gfCNCPoint4[10892] = {X 149.4831, Y 49.3200, Z -5.5000, A 0.000, B 0.000, C 0.000 }
gfCNCPoint4[10893] = {X 143.0396, Y 49.3200, Z -5.5000, A 0.000, B 0.000, C 0.000 }
gfCNCPoint4[10894] = {X 142.0831, Y 49.2128, Z -5.5000, A 0.000, B 0.000, C 0.000 }
gfCNCPoint4[10895] = {X 141.1741, Y 48.8964, Z -5.5000, A 0.000, B 0.000, C 0.000 }
gfCNCPoint4[10896] = {X 140.3576, Y 48.3866, Z -5.5000, A 0.000, B 0.000, C 0.000 }
gfCNCPoint4[10897] = {X 139.6743, Y 47.7087, Z -5.5000, A 0.000, B 0.000, C 0.000 }
gfCNCPoint4[10898] = {X 139.1581, Y 46.8964, Z -5.5000, A 0.000, B 0.000, C 0.000 }
gfCNCPoint4[10899] = {X 138.8346, Y 45.9899, Z -5.5000, A 0.000, B 0.000, C 0.000 }
gfCNCPoint4[10900] = {X 138.7198, Y 45.0342, Z -5.5000, A 0.000, B 0.000, C 0.000 }
gfCNCPoint4[10901] = {X 138.7200, Y 44.1494, Z -5.5000, A 0.000, B 0.000, C 0.000 }
gfCNCPoint4[10902] = {X 138.8305, Y 43.2364, Z -5.5000, A 0.000, B 0.000, C 0.000 }
gfCNCPoint4[10903] = {X 139.1317, Y 42.3675, Z -5.5000, A 0.000, B 0.000, C 0.000 }
gfCNCPoint4[10904] = {X 139.6099, Y 41.5821, Z -5.5000, A 0.000, B 0.000, C 0.000 }
gfCNCPoint4[10905] = {X 140.2436, Y 40.9157, Z -5.5000, A 0.000, B 0.000, C 0.000 }
gfCNCPoint4[10906] = {X 140.2436, Y 30.3967, Z -5.5000, A 0.000, B 0.000, C 0.000 }
gfCNCPoint4[10907] = {X 136.2436, Y 30.3967, Z -5.5000, A 0.000, B 0.000, C 0.000 }
gfCNCPoint4[10908] = {X 140.3236, Y 30.3967, Z -5.5000, A 0.000, B 0.000, C 0.000 }
gfCNCPoint4[10909] = {X 140.3236, Y 19.7977, Z -5.5000, A 0.000, B 0.000, C 0.000 }
gfCNCPoint4[10910] = {X 137.3795, Y 19.7972, Z -5.5000, A 0.000, B 0.000, C 0.000 }
gfCNCPoint4[10911] = {X 137.3567, Y 19.8337, Z -5.5000, A 0.000, B 0.000, C 0.000 }
gfCNCPoint4[10912] = {X 136.8341, Y 20.4660, Z -5.5000, A 0.000, B 0.000, C 0.000 }
gfCNCPoint4[10913] = {X 136.1996, Y 20.9859, Z -5.5000, A 0.000, B 0.000, C 0.000 }
gfCNCPoint4[10914] = {X 135.4768, Y 21.3738, Z -5.5000, A 0.000, B 0.000, C 0.000 }
gfCNCPoint4[10915] = {X 134.6929, Y 21.6153, Z -5.5000, A 0.000, B 0.000, C 0.000 }
gfCNCPoint4[10916] = {X 133.8772, Y 21.7014, Z -5.5000, A 0.000, B 0.000, C 0.000 }
gfCNCPoint4[10917] = {X 133.2006, Y 21.7015, Z -5.5000, A 0.000, B 0.000, C 0.000 }
gfCNCPoint4[10918] = {X 132.2572, Y 21.5952, Z -5.5000, A 0.000, B 0.000, C 0.000 }
gfCNCPoint4[10919] = {X 131.3610, Y 21.2816, Z -5.5000, A 0.000, B 0.000, C 0.000 }
gfCNCPoint4[10920] = {X 130.5570, Y 20.7765, Z -5.5000, A 0.000, B 0.000, C 0.000 }
gfCNCPoint4[10921] = {X 129.8857, Y 20.1051, Z -5.5000, A 0.000, B 0.000, C 0.000 }
gfCNCPoint4[10922] = {X 129.3805, Y 19.3012, Z -5.5000, A 0.000, B 0.000, C 0.000 }
gfCNCPoint4[10923] = {X 129.0669, Y 18.4050, Z -5.5000, A 0.000, B 0.000, C 0.000 }
gfCNCPoint4[10924] = {X 128.9606, Y 17.4615, Z -5.5000, A 0.000, B 0.000, C 0.000 }
gfCNCPoint4[10925] = {X 128.9606, Y 10.4835, Z -5.5000, A 0.000, B 0.000, C 0.000 }
gfCNCPoint4[10926] = {X 129.0655, Y 9.5466, Z -5.5000, A 0.000, B 0.000, C 0.000 }
gfCNCPoint4[10927] = {X 129.3747, Y 8.6559, Z -5.5000, A 0.000, B 0.000, C 0.000 }
gfCNCPoint4[10928] = {X 129.8732, Y 7.8557, Z -5.5000, A 0.000, B 0.000, C 0.000 }
gfCNCPoint4[10929] = {X 130.5362, Y 7.1853, Z -5.5000, A 0.000, B 0.000, C 0.000 }
gfCNCPoint4[10930] = {X 131.3309, Y 6.6781, Z -5.5000, A 0.000, B 0.000, C 0.000 }
gfCNCPoint4[10931] = {X 132.2180, Y 6.3589, Z -5.5000, A 0.000, B 0.000, C 0.000 }
gfCNCPoint4[10932] = {X 133.1538, Y 6.2438, Z -5.5000, A 0.000, B 0.000, C 0.000 }
gfCNCPoint4[10933] = {X 133.8858, Y 6.2437, Z -5.5000, A 0.000, B 0.000, C 0.000 }
gfCNCPoint4[10934] = {X 134.7031, Y 6.3318, Z -5.5000, A 0.000, B 0.000, C 0.000 }
gfCNCPoint4[10935] = {X 135.4881, Y 6.5760, Z -5.5000, A 0.000, B 0.000, C 0.000 }
gfCNCPoint4[10936] = {X 136.2112, Y 6.9670, Z -5.5000, A 0.000, B 0.000, C 0.000 }
gfCNCPoint4[10937] = {X 136.8453, Y 7.4903, Z -5.5000, A 0.000, B 0.000, C 0.000 }
gfCNCPoint4[10938] = {X 137.3665, Y 8.1260, Z -5.5000, A 0.000, B 0.000, C 0.000 }
gfCNCPoint4[10939] = {X 155.1554, Y 8.1273, Z -5.5000, A 0.000, B 0.000, C 0.000 }
gfCNCPoint4[10940] = {X 155.6773, Y 7.4904, Z -5.5000, A 0.000, B 0.000, C 0.000 }
gfCNCPoint4[10941] = {X 156.3124, Y 6.9664, Z -5.5000, A 0.000, B 0.000, C 0.000 }
gfCNCPoint4[10942] = {X 157.0368, Y 6.5750, Z -5.5000, A 0.000, B 0.000, C 0.000 }
gfCNCPoint4[10943] = {X 157.8232, Y 6.3311, Z -5.5000, A 0.000, B 0.000, C 0.000 }
gfCNCPoint4[10944] = {X 158.6420, Y 6.2437, Z -5.5000, A 0.000, B 0.000, C 0.000 }
gfCNCPoint4[10945] = {X 159.3770, Y 6.2439, Z -5.5000, A 0.000, B 0.000, C 0.000 }
gfCNCPoint4[10946] = {X 160.3114, Y 6.3606, Z -5.5000, A 0.000, B 0.000, C 0.000 }
gfCNCPoint4[10947] = {X 161.1970, Y 6.6806, Z -5.5000, A 0.000, B 0.000, C 0.000 }
gfCNCPoint4[10948] = {X 161.9902, Y 7.1882, Z -5.5000, A 0.000, B 0.000, C 0.000 }
gfCNCPoint4[10949] = {X 162.6517, Y 7.8584, Z -5.5000, A 0.000, B 0.000, C 0.000 }
gfCNCPoint4[10950] = {X 163.1490, Y 8.6580, Z -5.5000, A 0.000, B 0.000, C 0.000 }
gfCNCPoint4[10951] = {X 163.4575, Y 9.5477, Z -5.5000, A 0.000, B 0.000, C 0.000 }
gfCNCPoint4[10952] = {X 163.5621, Y 10.4835, Z -5.5000, A 0.000, B 0.000, C 0.000 }
gfCNCPoint4[10953] = {X 163.5621, Y 17.4615, Z -5.5000, A 0.000, B 0.000, C 0.000 }
gfCNCPoint4[10954] = {X 163.4575, Y 18.3975, Z -5.5000, A 0.000, B 0.000, C 0.000 }
gfCNCPoint4[10955] = {X 163.1489, Y 19.2873, Z -5.5000, A 0.000, B 0.000, C 0.000 }
gfCNCPoint4[10956] = {X 162.6514, Y 20.0870, Z -5.5000, A 0.000, B 0.000, C 0.000 }
gfCNCPoint4[10957] = {X 161.9897, Y 20.7572, Z -5.5000, A 0.000, B 0.000, C 0.000 }
gfCNCPoint4[10958] = {X 161.1964, Y 21.2648, Z -5.5000, A 0.000, B 0.000, C 0.000 }
gfCNCPoint4[10959] = {X 160.3106, Y 21.5847, Z -5.5000, A 0.000, B 0.000, C 0.000 }
gfCNCPoint4[10960] = {X 159.3760, Y 21.7012, Z -5.5000, A 0.000, B 0.000, C 0.000 }
gfCNCPoint4[10961] = {X 158.6796, Y 21.7015, Z -5.5000, A 0.000, B 0.000, C 0.000 }
gfCNCPoint4[10962] = {X 157.8483, Y 21.6166, Z -5.5000, A 0.000, B 0.000, C 0.000 }
gfCNCPoint4[10963] = {X 157.0495, Y 21.3715, Z -5.5000, A 0.000, B 0.000, C 0.000 }
gfCNCPoint4[10964] = {X 156.3137, Y 20.9756, Z -5.5000, A 0.000, B 0.000, C 0.000 }
gfCNCPoint4[10965] = {X 155.6689, Y 20.4441, Z -5.5000, A 0.000, B 0.000, C 0.000 }
gfCNCPoint4[10966] = {X 155.1400, Y 19.7973, Z -5.5000, A 0.000, B 0.000, C 0.000 }
gfCNCPoint4[10967] = {X 152.1967, Y 19.7984, Z -5.5000, A 0.000, B 0.000, C 0.000 }
gfCNCPoint4[10968] = {X 152.1954, Y 40.9056, Z -5.5000, A 0.000, B 0.000, C 0.000 }
gfCNCPoint4[10969] = {X 152.6809, Y 41.4282, Z -5.5000, A 0.000, B 0.000, C 0.000 }
gfCNCPoint4[10970] = {X 152.7744, Y 41.5396, Z -5.5000, A 0.000, B 0.000, C 0.000 }
gfCNCPoint4[10971] = {X 153.2900, Y 42.3496, Z -5.5000, A 0.000, B 0.000, C 0.000 }
gfCNCPoint4[10972] = {X 153.6117, Y 43.2543, Z -5.5000, A 0.000, B 0.000, C 0.000 }
gfCNCPoint4[10973] = {X 153.7231, Y 44.2080, Z -5.5000, A 0.000, B 0.000, C 0.000 }
gfCNCPoint4[10974] = {X 153.7229, Y 45.0408, Z -5.5000, A 0.000, B 0.000, C 0.000 }
gfCNCPoint4[10975] = {X 153.6089, Y 45.9775, Z -5.5000, A 0.000, B 0.000, C 0.000 }
gfCNCPoint4[10976] = {X 153.2905, Y 46.8659, Z -5.5000, A 0.000, B 0.000, C 0.000 }
gfCNCPoint4[10977] = {X 152.7835, Y 47.6618, Z -5.5000, A 0.000, B 0.000, C 0.000 }
gfCNCPoint4[10978] = {X 152.1130, Y 48.3258, Z -5.5000, A 0.000, B 0.000, C 0.000 }
gfCNCPoint4[10979] = {X 151.3123, Y 48.8251, Z -5.5000, A 0.000, B 0.000, C 0.000 }
gfCNCPoint4[10980] = {X 150.4209, Y 49.1350, Z -5.5000, A 0.000, B 0.000, C 0.000 }
gfCNCPoint4[10981] = {X 149.4831, Y 49.2400, Z -5.5000, A 0.000, B 0.000, C 0.000 }
gfCNCPoint4[10982] = {X 143.0396, Y 49.2400, Z -5.5000, A 0.000, B 0.000, C 0.000 }
gfCNCPoint4[10983] = {X 142.1008, Y 49.1348, Z -5.5000, A 0.000, B 0.000, C 0.000 }
gfCNCPoint4[10984] = {X 141.2086, Y 48.8243, Z -5.5000, A 0.000, B 0.000, C 0.000 }
gfCNCPoint4[10985] = {X 140.4073, Y 48.3239, Z -5.5000, A 0.000, B 0.000, C 0.000 }
gfCNCPoint4[10986] = {X 139.7367, Y 47.6586, Z -5.5000, A 0.000, B 0.000, C 0.000 }
gfCNCPoint4[10987] = {X 139.2300, Y 46.8612, Z -5.5000, A 0.000, B 0.000, C 0.000 }
gfCNCPoint4[10988] = {X 138.9124, Y 45.9715, Z -5.5000, A 0.000, B 0.000, C 0.000 }
gfCNCPoint4[10989] = {X 138.7998, Y 45.0336, Z -5.5000, A 0.000, B 0.000, C 0.000 }
gfCNCPoint4[10990] = {X 138.8000, Y 44.1505, Z -5.5000, A 0.000, B 0.000, C 0.000 }
gfCNCPoint4[10991] = {X 138.9105, Y 43.2454, Z -5.5000, A 0.000, B 0.000, C 0.000 }
gfCNCPoint4[10992] = {X 139.2119, Y 42.3850, Z -5.5000, A 0.000, B 0.000, C 0.000 }
gfCNCPoint4[10993] = {X 139.6903, Y 41.6088, Z -5.5000, A 0.000, B 0.000, C 0.000 }
gfCNCPoint4[10994] = {X 140.3236, Y 40.9529, Z -5.5000, A 0.000, B 0.000, C 0.000 }
gfCNCPoint4[10995] = {X 140.3236, Y 30.3967, Z -5.5000, A 0.000, B 0.000, C 0.000 }
gfCNCPoint4[10996] = {X 136.3236, Y 30.3967, Z -5.5000, A 0.000, B 0.000, C 0.000 }
gfCNCPoint4[10997] = {X 140.4036, Y 30.3967, Z -5.5000, A 0.000, B 0.000, C 0.000 }
gfCNCPoint4[10998] = {X 140.4036, Y 19.7178, Z -5.5000, A 0.000, B 0.000, C 0.000 }
gfCNCPoint4[10999] = {X 137.3353, Y 19.7172, Z -5.5000, A 0.000, B 0.000, C 0.000 }
gfCNCPoint4[11000] = {X 137.2896, Y 19.7900, Z -5.5000, A 0.000, B 0.000, C 0.000 }
gfCNCPoint4[11001] = {X 136.7769, Y 20.4101, Z -5.5000, A 0.000, B 0.000, C 0.000 }
gfCNCPoint4[11002] = {X 136.1544, Y 20.9198, Z -5.5000, A 0.000, B 0.000, C 0.000 }
gfCNCPoint4[11003] = {X 135.4455, Y 21.3002, Z -5.5000, A 0.000, B 0.000, C 0.000 }
gfCNCPoint4[11004] = {X 134.6766, Y 21.5370, Z -5.5000, A 0.000, B 0.000, C 0.000 }
gfCNCPoint4[11005] = {X 133.8765, Y 21.6214, Z -5.5000, A 0.000, B 0.000, C 0.000 }
gfCNCPoint4[11006] = {X 133.2006, Y 21.6215, Z -5.5000, A 0.000, B 0.000, C 0.000 }
gfCNCPoint4[11007] = {X 132.2750, Y 21.5172, Z -5.5000, A 0.000, B 0.000, C 0.000 }
gfCNCPoint4[11008] = {X 131.3957, Y 21.2096, Z -5.5000, A 0.000, B 0.000, C 0.000 }
gfCNCPoint4[11009] = {X 130.6069, Y 20.7140, Z -5.5000, A 0.000, B 0.000, C 0.000 }
gfCNCPoint4[11010] = {X 129.9482, Y 20.0553, Z -5.5000, A 0.000, B 0.000, C 0.000 }
gfCNCPoint4[11011] = {X 129.4526, Y 19.2665, Z -5.5000, A 0.000, B 0.000, C 0.000 }
gfCNCPoint4[11012] = {X 129.1449, Y 18.3872, Z -5.5000, A 0.000, B 0.000, C 0.000 }
gfCNCPoint4[11013] = {X 129.0406, Y 17.4615, Z -5.5000, A 0.000, B 0.000, C 0.000 }
gfCNCPoint4[11014] = {X 129.0406, Y 10.4835, Z -5.5000, A 0.000, B 0.000, C 0.000 }
gfCNCPoint4[11015] = {X 129.1435, Y 9.5642, Z -5.5000, A 0.000, B 0.000, C 0.000 }
gfCNCPoint4[11016] = {X 129.4469, Y 8.6904, Z -5.5000, A 0.000, B 0.000, C 0.000 }
gfCNCPoint4[11017] = {X 129.9360, Y 7.9052, Z -5.5000, A 0.000, B 0.000, C 0.000 }
gfCNCPoint4[11018] = {X 130.5864, Y 7.2475, Z -5.5000, A 0.000, B 0.000, C 0.000 }
gfCNCPoint4[11019] = {X 131.3661, Y 6.7499, Z -5.5000, A 0.000, B 0.000, C 0.000 }
gfCNCPoint4[11020] = {X 132.2366, Y 6.4368, Z -5.5000, A 0.000, B 0.000, C 0.000 }
gfCNCPoint4[11021] = {X 133.1547, Y 6.3238, Z -5.5000, A 0.000, B 0.000, C 0.000 }
gfCNCPoint4[11022] = {X 133.8850, Y 6.3237, Z -5.5000, A 0.000, B 0.000, C 0.000 }
gfCNCPoint4[11023] = {X 134.6952, Y 6.4119, Z -5.5000, A 0.000, B 0.000, C 0.000 }
gfCNCPoint4[11024] = {X 135.4728, Y 6.6563, Z -5.5000, A 0.000, B 0.000, C 0.000 }
gfCNCPoint4[11025] = {X 136.1877, Y 7.0477, Z -5.5000, A 0.000, B 0.000, C 0.000 }
gfCNCPoint4[11026] = {X 136.8126, Y 7.5710, Z -5.5000, A 0.000, B 0.000, C 0.000 }
gfCNCPoint4[11027] = {X 137.3235, Y 8.2060, Z -5.5000, A 0.000, B 0.000, C 0.000 }
gfCNCPoint4[11028] = {X 155.1984, Y 8.2073, Z -5.5000, A 0.000, B 0.000, C 0.000 }
gfCNCPoint4[11029] = {X 155.7100, Y 7.5711, Z -5.5000, A 0.000, B 0.000, C 0.000 }
gfCNCPoint4[11030] = {X 156.3359, Y 7.0471, Z -5.5000, A 0.000, B 0.000, C 0.000 }
gfCNCPoint4[11031] = {X 157.0521, Y 6.6554, Z -5.5000, A 0.000, B 0.000, C 0.000 }
gfCNCPoint4[11032] = {X 157.8310, Y 6.4111, Z -5.5000, A 0.000, B 0.000, C 0.000 }
gfCNCPoint4[11033] = {X 158.6427, Y 6.3237, Z -5.5000, A 0.000, B 0.000, C 0.000 }
gfCNCPoint4[11034] = {X 159.3760, Y 6.3239, Z -5.5000, A 0.000, B 0.000, C 0.000 }
gfCNCPoint4[11035] = {X 160.2928, Y 6.4383, Z -5.5000, A 0.000, B 0.000, C 0.000 }
gfCNCPoint4[11036] = {X 161.1617, Y 6.7524, Z -5.5000, A 0.000, B 0.000, C 0.000 }
gfCNCPoint4[11037] = {X 161.9398, Y 7.2504, Z -5.5000, A 0.000, B 0.000, C 0.000 }
gfCNCPoint4[11038] = {X 162.5889, Y 7.9079, Z -5.5000, A 0.000, B 0.000, C 0.000 }
gfCNCPoint4[11039] = {X 163.0768, Y 8.6925, Z -5.5000, A 0.000, B 0.000, C 0.000 }
gfCNCPoint4[11040] = {X 163.3795, Y 9.5653, Z -5.5000, A 0.000, B 0.000, C 0.000 }
gfCNCPoint4[11041] = {X 163.4821, Y 10.4835, Z -5.5000, A 0.000, B 0.000, C 0.000 }
gfCNCPoint4[11042] = {X 163.4821, Y 17.4615, Z -5.5000, A 0.000, B 0.000, C 0.000 }
gfCNCPoint4[11043] = {X 163.3795, Y 18.3798, Z -5.5000, A 0.000, B 0.000, C 0.000 }
gfCNCPoint4[11044] = {X 163.0767, Y 19.2527, Z -5.5000, A 0.000, B 0.000, C 0.000 }
gfCNCPoint4[11045] = {X 162.5887, Y 20.0373, Z -5.5000, A 0.000, B 0.000, C 0.000 }
gfCNCPoint4[11046] = {X 161.9396, Y 20.6948, Z -5.5000, A 0.000, B 0.000, C 0.000 }
gfCNCPoint4[11047] = {X 161.1613, Y 21.1929, Z -5.5000, A 0.000, B 0.000, C 0.000 }
gfCNCPoint4[11048] = {X 160.2923, Y 21.5068, Z -5.5000, A 0.000, B 0.000, C 0.000 }
gfCNCPoint4[11049] = {X 159.3755, Y 21.6212, Z -5.5000, A 0.000, B 0.000, C 0.000 }
gfCNCPoint4[11050] = {X 158.6799, Y 21.6215, Z -5.5000, A 0.000, B 0.000, C 0.000 }
gfCNCPoint4[11051] = {X 157.8558, Y 21.5365, Z -5.5000, A 0.000, B 0.000, C 0.000 }
gfCNCPoint4[11052] = {X 157.0646, Y 21.2910, Z -5.5000, A 0.000, B 0.000, C 0.000 }
gfCNCPoint4[11053] = {X 156.3370, Y 20.8948, Z -5.5000, A 0.000, B 0.000, C 0.000 }
gfCNCPoint4[11054] = {X 155.7016, Y 20.3633, Z -5.5000, A 0.000, B 0.000, C 0.000 }
gfCNCPoint4[11055] = {X 155.1830, Y 19.7172, Z -5.5000, A 0.000, B 0.000, C 0.000 }
gfCNCPoint4[11056] = {X 152.1167, Y 19.7184, Z -5.5000, A 0.000, B 0.000, C 0.000 }
gfCNCPoint4[11057] = {X 152.1154, Y 40.9370, Z -5.5000, A 0.000, B 0.000, C 0.000 }
gfCNCPoint4[11058] = {X 152.6209, Y 41.4812, Z -5.5000, A 0.000, B 0.000, C 0.000 }
gfCNCPoint4[11059] = {X 152.7126, Y 41.5905, Z -5.5000, A 0.000, B 0.000, C 0.000 }
gfCNCPoint4[11060] = {X 153.2184, Y 42.3852, Z -5.5000, A 0.000, B 0.000, C 0.000 }
gfCNCPoint4[11061] = {X 153.5338, Y 43.2727, Z -5.5000, A 0.000, B 0.000, C 0.000 }
gfCNCPoint4[11062] = {X 153.6431, Y 44.2083, Z -5.5000, A 0.000, B 0.000, C 0.000 }
gfCNCPoint4[11063] = {X 153.6429, Y 45.0400, Z -5.5000, A 0.000, B 0.000, C 0.000 }
gfCNCPoint4[11064] = {X 153.5310, Y 45.9591, Z -5.5000, A 0.000, B 0.000, C 0.000 }
gfCNCPoint4[11065] = {X 153.2186, Y 46.8306, Z -5.5000, A 0.000, B 0.000, C 0.000 }
gfCNCPoint4[11066] = {X 152.7212, Y 47.6115, Z -5.5000, A 0.000, B 0.000, C 0.000 }
gfCNCPoint4[11067] = {X 152.0634, Y 48.2631, Z -5.5000, A 0.000, B 0.000, C 0.000 }
gfCNCPoint4[11068] = {X 151.2778, Y 48.7530, Z -5.5000, A 0.000, B 0.000, C 0.000 }
gfCNCPoint4[11069] = {X 150.4032, Y 49.0570, Z -5.5000, A 0.000, B 0.000, C 0.000 }
gfCNCPoint4[11070] = {X 149.4831, Y 49.1600, Z -5.5000, A 0.000, B 0.000, C 0.000 }
gfCNCPoint4[11071] = {X 143.0396, Y 49.1600, Z -5.5000, A 0.000, B 0.000, C 0.000 }
gfCNCPoint4[11072] = {X 142.1185, Y 49.0567, Z -5.5000, A 0.000, B 0.000, C 0.000 }
gfCNCPoint4[11073] = {X 141.2432, Y 48.7521, Z -5.5000, A 0.000, B 0.000, C 0.000 }
gfCNCPoint4[11074] = {X 140.4570, Y 48.2612, Z -5.5000, A 0.000, B 0.000, C 0.000 }
gfCNCPoint4[11075] = {X 139.7990, Y 47.6084, Z -5.5000, A 0.000, B 0.000, C 0.000 }
gfCNCPoint4[11076] = {X 139.3019, Y 46.8261, Z -5.5000, A 0.000, B 0.000, C 0.000 }
gfCNCPoint4[11077] = {X 138.9903, Y 45.9532, Z -5.5000, A 0.000, B 0.000, C 0.000 }
gfCNCPoint4[11078] = {X 138.8798, Y 45.0329, Z -5.5000, A 0.000, B 0.000, C 0.000 }
gfCNCPoint4[11079] = {X 138.8800, Y 44.1516, Z -5.5000, A 0.000, B 0.000, C 0.000 }
gfCNCPoint4[11080] = {X 138.9906, Y 43.2545, Z -5.5000, A 0.000, B 0.000, C 0.000 }
gfCNCPoint4[11081] = {X 139.2922, Y 42.4026, Z -5.5000, A 0.000, B 0.000, C 0.000 }
gfCNCPoint4[11082] = {X 139.7708, Y 41.6358, Z -5.5000, A 0.000, B 0.000, C 0.000 }
gfCNCPoint4[11083] = {X 140.4036, Y 40.9906, Z -5.5000, A 0.000, B 0.000, C 0.000 }
gfCNCPoint4[11084] = {X 140.4036, Y 30.3967, Z -5.5000, A 0.000, B 0.000, C 0.000 }
gfCNCPoint4[11085] = {X 136.4036, Y 30.3967, Z -5.5000, A 0.000, B 0.000, C 0.000 }
gfCNCPoint4[11086] = {X 140.4836, Y 30.3967, Z -5.5000, A 0.000, B 0.000, C 0.000 }
gfCNCPoint4[11087] = {X 140.4836, Y 19.6378, Z -5.5000, A 0.000, B 0.000, C 0.000 }
gfCNCPoint4[11088] = {X 137.2910, Y 19.6372, Z -5.5000, A 0.000, B 0.000, C 0.000 }
gfCNCPoint4[11089] = {X 137.2218, Y 19.7475, Z -5.5000, A 0.000, B 0.000, C 0.000 }
gfCNCPoint4[11090] = {X 136.5756, Y 20.4907, Z -5.5000, A 0.000, B 0.000, C 0.000 }
gfCNCPoint4[11091] = {X 135.7702, Y 21.0573, Z -5.5000, A 0.000, B 0.000, C 0.000 }
gfCNCPoint4[11092] = {X 134.8524, Y 21.4145, Z -5.5000, A 0.000, B 0.000, C 0.000 }
gfCNCPoint4[11093] = {X 133.8758, Y 21.5414, Z -5.5000, A 0.000, B 0.000, C 0.000 }
gfCNCPoint4[11094] = {X 133.2006, Y 21.5415, Z -5.5000, A 0.000, B 0.000, C 0.000 }
gfCNCPoint4[11095] = {X 132.2928, Y 21.4392, Z -5.5000, A 0.000, B 0.000, C 0.000 }
gfCNCPoint4[11096] = {X 131.4304, Y 21.1375, Z -5.5000, A 0.000, B 0.000, C 0.000 }
gfCNCPoint4[11097] = {X 130.6568, Y 20.6514, Z -5.5000, A 0.000, B 0.000, C 0.000 }
gfCNCPoint4[11098] = {X 130.0108, Y 20.0054, Z -5.5000, A 0.000, B 0.000, C 0.000 }
gfCNCPoint4[11099] = {X 129.5247, Y 19.2318, Z -5.5000, A 0.000, B 0.000, C 0.000 }
gfCNCPoint4[11100] = {X 129.2229, Y 18.3694, Z -5.5000, A 0.000, B 0.000, C 0.000 }
gfCNCPoint4[11101] = {X 129.1206, Y 17.4615, Z -5.5000, A 0.000, B 0.000, C 0.000 }
gfCNCPoint4[11102] = {X 129.1206, Y 10.4835, Z -5.5000, A 0.000, B 0.000, C 0.000 }
gfCNCPoint4[11103] = {X 129.2215, Y 9.5820, Z -5.5000, A 0.000, B 0.000, C 0.000 }
gfCNCPoint4[11104] = {X 129.5191, Y 8.7250, Z -5.5000, A 0.000, B 0.000, C 0.000 }
gfCNCPoint4[11105] = {X 129.9986, Y 7.9550, Z -5.5000, A 0.000, B 0.000, C 0.000 }
gfCNCPoint4[11106] = {X 130.6365, Y 7.3099, Z -5.5000, A 0.000, B 0.000, C 0.000 }
gfCNCPoint4[11107] = {X 131.4011, Y 6.8218, Z -5.5000, A 0.000, B 0.000, C 0.000 }
gfCNCPoint4[11108] = {X 132.2547, Y 6.5147, Z -5.5000, A 0.000, B 0.000, C 0.000 }
gfCNCPoint4[11109] = {X 133.1551, Y 6.4038, Z -5.5000, A 0.000, B 0.000, C 0.000 }
gfCNCPoint4[11110] = {X 133.8841, Y 6.4037, Z -5.5000, A 0.000, B 0.000, C 0.000 }
gfCNCPoint4[11111] = {X 134.6873, Y 6.4920, Z -5.5000, A 0.000, B 0.000, C 0.000 }
gfCNCPoint4[11112] = {X 135.4573, Y 6.7367, Z -5.5000, A 0.000, B 0.000, C 0.000 }
gfCNCPoint4[11113] = {X 136.1639, Y 7.1284, Z -5.5000, A 0.000, B 0.000, C 0.000 }
gfCNCPoint4[11114] = {X 136.7795, Y 7.6517, Z -5.5000, A 0.000, B 0.000, C 0.000 }
gfCNCPoint4[11115] = {X 137.2800, Y 8.2860, Z -5.5000, A 0.000, B 0.000, C 0.000 }
gfCNCPoint4[11116] = {X 155.2419, Y 8.2873, Z -5.5000, A 0.000, B 0.000, C 0.000 }
gfCNCPoint4[11117] = {X 155.2874, Y 8.2177, Z -5.5000, A 0.000, B 0.000, C 0.000 }
gfCNCPoint4[11118] = {X 155.3342, Y 8.1491, Z -5.5000, A 0.000, B 0.000, C 0.000 }
gfCNCPoint4[11119] = {X 155.9794, Y 7.4256, Z -5.5000, A 0.000, B 0.000, C 0.000 }
gfCNCPoint4[11120] = {X 156.7770, Y 6.8747, Z -5.5000, A 0.000, B 0.000, C 0.000 }
gfCNCPoint4[11121] = {X 157.6820, Y 6.5276, Z -5.5000, A 0.000, B 0.000, C 0.000 }
gfCNCPoint4[11122] = {X 158.6434, Y 6.4037, Z -5.5000, A 0.000, B 0.000, C 0.000 }
gfCNCPoint4[11123] = {X 159.3750, Y 6.4039, Z -5.5000, A 0.000, B 0.000, C 0.000 }
gfCNCPoint4[11124] = {X 160.2741, Y 6.5161, Z -5.5000, A 0.000, B 0.000, C 0.000 }
gfCNCPoint4[11125] = {X 161.1263, Y 6.8241, Z -5.5000, A 0.000, B 0.000, C 0.000 }
gfCNCPoint4[11126] = {X 161.8895, Y 7.3126, Z -5.5000, A 0.000, B 0.000, C 0.000 }
gfCNCPoint4[11127] = {X 162.5260, Y 7.9574, Z -5.5000, A 0.000, B 0.000, C 0.000 }
gfCNCPoint4[11128] = {X 163.0046, Y 8.7269, Z -5.5000, A 0.000, B 0.000, C 0.000 }
gfCNCPoint4[11129] = {X 163.3015, Y 9.5830, Z -5.5000, A 0.000, B 0.000, C 0.000 }
gfCNCPoint4[11130] = {X 163.4021, Y 10.4835, Z -5.5000, A 0.000, B 0.000, C 0.000 }
gfCNCPoint4[11131] = {X 163.4021, Y 17.4615, Z -5.5000, A 0.000, B 0.000, C 0.000 }
gfCNCPoint4[11132] = {X 163.3015, Y 18.3621, Z -5.5000, A 0.000, B 0.000, C 0.000 }
gfCNCPoint4[11133] = {X 163.0046, Y 19.2182, Z -5.5000, A 0.000, B 0.000, C 0.000 }
gfCNCPoint4[11134] = {X 162.5260, Y 19.9876, Z -5.5000, A 0.000, B 0.000, C 0.000 }
gfCNCPoint4[11135] = {X 161.8895, Y 20.6325, Z -5.5000, A 0.000, B 0.000, C 0.000 }
gfCNCPoint4[11136] = {X 161.1263, Y 21.1209, Z -5.5000, A 0.000, B 0.000, C 0.000 }
gfCNCPoint4[11137] = {X 160.2741, Y 21.4289, Z -5.5000, A 0.000, B 0.000, C 0.000 }
gfCNCPoint4[11138] = {X 159.3750, Y 21.5412, Z -5.5000, A 0.000, B 0.000, C 0.000 }
gfCNCPoint4[11139] = {X 158.6802, Y 21.5415, Z -5.5000, A 0.000, B 0.000, C 0.000 }
gfCNCPoint4[11140] = {X 157.8634, Y 21.4563, Z -5.5000, A 0.000, B 0.000, C 0.000 }
gfCNCPoint4[11141] = {X 157.0798, Y 21.2106, Z -5.5000, A 0.000, B 0.000, C 0.000 }
gfCNCPoint4[11142] = {X 156.3607, Y 20.8140, Z -5.5000, A 0.000, B 0.000, C 0.000 }
gfCNCPoint4[11143] = {X 155.7346, Y 20.2825, Z -5.5000, A 0.000, B 0.000, C 0.000 }
gfCNCPoint4[11144] = {X 155.2267, Y 19.6372, Z -5.5000, A 0.000, B 0.000, C 0.000 }
gfCNCPoint4[11145] = {X 152.0367, Y 19.6385, Z -5.5000, A 0.000, B 0.000, C 0.000 }
gfCNCPoint4[11146] = {X 152.0354, Y 40.9684, Z -5.5000, A 0.000, B 0.000, C 0.000 }
gfCNCPoint4[11147] = {X 152.5609, Y 41.5342, Z -5.5000, A 0.000, B 0.000, C 0.000 }
gfCNCPoint4[11148] = {X 152.6509, Y 41.6413, Z -5.5000, A 0.000, B 0.000, C 0.000 }
gfCNCPoint4[11149] = {X 153.1467, Y 42.4207, Z -5.5000, A 0.000, B 0.000, C 0.000 }
gfCNCPoint4[11150] = {X 153.4560, Y 43.2911, Z -5.5000, A 0.000, B 0.000, C 0.000 }
gfCNCPoint4[11151] = {X 153.5631, Y 44.2086, Z -5.5000, A 0.000, B 0.000, C 0.000 }
gfCNCPoint4[11152] = {X 153.5629, Y 45.0392, Z -5.5000, A 0.000, B 0.000, C 0.000 }
gfCNCPoint4[11153] = {X 153.4532, Y 45.9406, Z -5.5000, A 0.000, B 0.000, C 0.000 }
gfCNCPoint4[11154] = {X 153.1468, Y 46.7954, Z -5.5000, A 0.000, B 0.000, C 0.000 }
gfCNCPoint4[11155] = {X 152.6589, Y 47.5613, Z -5.5000, A 0.000, B 0.000, C 0.000 }
gfCNCPoint4[11156] = {X 152.0138, Y 48.2003, Z -5.5000, A 0.000, B 0.000, C 0.000 }
gfCNCPoint4[11157] = {X 151.2432, Y 48.6808, Z -5.5000, A 0.000, B 0.000, C 0.000 }
gfCNCPoint4[11158] = {X 150.3855, Y 48.9789, Z -5.5000, A 0.000, B 0.000, C 0.000 }
gfCNCPoint4[11159] = {X 149.4831, Y 49.0800, Z -5.5000, A 0.000, B 0.000, C 0.000 }
gfCNCPoint4[11160] = {X 143.0396, Y 49.0800, Z -5.5000, A 0.000, B 0.000, C 0.000 }
gfCNCPoint4[11161] = {X 142.1362, Y 48.9787, Z -5.5000, A 0.000, B 0.000, C 0.000 }
gfCNCPoint4[11162] = {X 141.2777, Y 48.6799, Z -5.5000, A 0.000, B 0.000, C 0.000 }
gfCNCPoint4[11163] = {X 140.5066, Y 48.1985, Z -5.5000, A 0.000, B 0.000, C 0.000 }
gfCNCPoint4[11164] = {X 139.8613, Y 47.5582, Z -5.5000, A 0.000, B 0.000, C 0.000 }
gfCNCPoint4[11165] = {X 139.3737, Y 46.7910, Z -5.5000, A 0.000, B 0.000, C 0.000 }
gfCNCPoint4[11166] = {X 139.0682, Y 45.9349, Z -5.5000, A 0.000, B 0.000, C 0.000 }
gfCNCPoint4[11167] = {X 138.9598, Y 45.0323, Z -5.5000, A 0.000, B 0.000, C 0.000 }
gfCNCPoint4[11168] = {X 138.9600, Y 44.1527, Z -5.5000, A 0.000, B 0.000, C 0.000 }
gfCNCPoint4[11169] = {X 139.0706, Y 43.2637, Z -5.5000, A 0.000, B 0.000, C 0.000 }
gfCNCPoint4[11170] = {X 139.3725, Y 42.4203, Z -5.5000, A 0.000, B 0.000, C 0.000 }
gfCNCPoint4[11171] = {X 139.8512, Y 41.6631, Z -5.5000, A 0.000, B 0.000, C 0.000 }
gfCNCPoint4[11172] = {X 140.4836, Y 41.0287, Z -5.5000, A 0.000, B 0.000, C 0.000 }
gfCNCPoint4[11173] = {X 140.4836, Y 30.3967, Z -5.5000, A 0.000, B 0.000, C 0.000 }
gfCNCPoint4[11174] = {X 136.4836, Y 30.3967, Z -5.5000, A 0.000, B 0.000, C 0.000 }
gfCNCPoint4[11175] = {X 140.5636, Y 30.3967, Z -5.5000, A 0.000, B 0.000, C 0.000 }
gfCNCPoint4[11176] = {X 140.5636, Y 19.9577, Z -5.5000, A 0.000, B 0.000, C 0.000 }
gfCNCPoint4[11177] = {X 140.5640, Y 19.5578, Z -5.5000, A 0.000, B 0.000, C 0.000 }
gfCNCPoint4[11178] = {X 137.2663, Y 19.5572, Z -5.5000, A 0.000, B 0.000, C 0.000 }
gfCNCPoint4[11179] = {X 137.2442, Y 19.5612, Z -5.5000, A 0.000, B 0.000, C 0.000 }
gfCNCPoint4[11180] = {X 137.1366, Y 19.7304, Z -5.5000, A 0.000, B 0.000, C 0.000 }
gfCNCPoint4[11181] = {X 136.4971, Y 20.4535, Z -5.5000, A 0.000, B 0.000, C 0.000 }
gfCNCPoint4[11182] = {X 135.7030, Y 21.0024, Z -5.5000, A 0.000, B 0.000, C 0.000 }
gfCNCPoint4[11183] = {X 134.8005, Y 21.3451, Z -5.5000, A 0.000, B 0.000, C 0.000 }
gfCNCPoint4[11184] = {X 133.8422, Y 21.4615, Z -5.5000, A 0.000, B 0.000, C 0.000 }
gfCNCPoint4[11185] = {X 133.2006, Y 21.4615, Z -5.5000, A 0.000, B 0.000, C 0.000 }
gfCNCPoint4[11186] = {X 132.3106, Y 21.3612, Z -5.5000, A 0.000, B 0.000, C 0.000 }
gfCNCPoint4[11187] = {X 131.4651, Y 21.0654, Z -5.5000, A 0.000, B 0.000, C 0.000 }
gfCNCPoint4[11188] = {X 130.7067, Y 20.5889, Z -5.5000, A 0.000, B 0.000, C 0.000 }
gfCNCPoint4[11189] = {X 130.0733, Y 19.9555, Z -5.5000, A 0.000, B 0.000, C 0.000 }
gfCNCPoint4[11190] = {X 129.5968, Y 19.1971, Z -5.5000, A 0.000, B 0.000, C 0.000 }
gfCNCPoint4[11191] = {X 129.3009, Y 18.3516, Z -5.5000, A 0.000, B 0.000, C 0.000 }
gfCNCPoint4[11192] = {X 129.2006, Y 17.4615, Z -5.5000, A 0.000, B 0.000, C 0.000 }
gfCNCPoint4[11193] = {X 129.2006, Y 10.4835, Z -5.5000, A 0.000, B 0.000, C 0.000 }
gfCNCPoint4[11194] = {X 129.3009, Y 9.5934, Z -5.5000, A 0.000, B 0.000, C 0.000 }
gfCNCPoint4[11195] = {X 129.5968, Y 8.7480, Z -5.5000, A 0.000, B 0.000, C 0.000 }
gfCNCPoint4[11196] = {X 130.0733, Y 7.9896, Z -5.5000, A 0.000, B 0.000, C 0.000 }
gfCNCPoint4[11197] = {X 130.7067, Y 7.3562, Z -5.5000, A 0.000, B 0.000, C 0.000 }
gfCNCPoint4[11198] = {X 131.4651, Y 6.8796, Z -5.5000, A 0.000, B 0.000, C 0.000 }
gfCNCPoint4[11199] = {X 132.3106, Y 6.5838, Z -5.5000, A 0.000, B 0.000, C 0.000 }
gfCNCPoint4[11200] = {X 133.2007, Y 6.4835, Z -5.5000, A 0.000, B 0.000, C 0.000 }
gfCNCPoint4[11201] = {X 133.8833, Y 6.4837, Z -5.5000, A 0.000, B 0.000, C 0.000 }
gfCNCPoint4[11202] = {X 134.6792, Y 6.5721, Z -5.5000, A 0.000, B 0.000, C 0.000 }
gfCNCPoint4[11203] = {X 135.4416, Y 6.8171, Z -5.5000, A 0.000, B 0.000, C 0.000 }
gfCNCPoint4[11204] = {X 136.1399, Y 7.2092, Z -5.5000, A 0.000, B 0.000, C 0.000 }
gfCNCPoint4[11205] = {X 136.7461, Y 7.7325, Z -5.5000, A 0.000, B 0.000, C 0.000 }
gfCNCPoint4[11206] = {X 137.2359, Y 8.3660, Z -5.5000, A 0.000, B 0.000, C 0.000 }
gfCNCPoint4[11207] = {X 155.2276, Y 8.3660, Z -5.5000, A 0.000, B 0.000, C 0.000 }
gfCNCPoint4[11208] = {X 155.2814, Y 8.3748, Z -5.5000, A 0.000, B 0.000, C 0.000 }
gfCNCPoint4[11209] = {X 155.3394, Y 8.2840, Z -5.5000, A 0.000, B 0.000, C 0.000 }
gfCNCPoint4[11210] = {X 155.3998, Y 8.1949, Z -5.5000, A 0.000, B 0.000, C 0.000 }
gfCNCPoint4[11211] = {X 156.0392, Y 7.4796, Z -5.5000, A 0.000, B 0.000, C 0.000 }
gfCNCPoint4[11212] = {X 156.8304, Y 6.9370, Z -5.5000, A 0.000, B 0.000, C 0.000 }
gfCNCPoint4[11213] = {X 157.7281, Y 6.5985, Z -5.5000, A 0.000, B 0.000, C 0.000 }
gfCNCPoint4[11214] = {X 158.6806, Y 6.4835, Z -5.5000, A 0.000, B 0.000, C 0.000 }
gfCNCPoint4[11215] = {X 159.3739, Y 6.4839, Z -5.5000, A 0.000, B 0.000, C 0.000 }
gfCNCPoint4[11216] = {X 160.2554, Y 6.5939, Z -5.5000, A 0.000, B 0.000, C 0.000 }
gfCNCPoint4[11217] = {X 161.0909, Y 6.8959, Z -5.5000, A 0.000, B 0.000, C 0.000 }
gfCNCPoint4[11218] = {X 161.8391, Y 7.3747, Z -5.5000, A 0.000, B 0.000, C 0.000 }
gfCNCPoint4[11219] = {X 162.4632, Y 8.0070, Z -5.5000, A 0.000, B 0.000, C 0.000 }
gfCNCPoint4[11220] = {X 162.9324, Y 8.7613, Z -5.5000, A 0.000, B 0.000, C 0.000 }
gfCNCPoint4[11221] = {X 163.2234, Y 9.6007, Z -5.5000, A 0.000, B 0.000, C 0.000 }
gfCNCPoint4[11222] = {X 163.3221, Y 10.4835, Z -5.5000, A 0.000, B 0.000, C 0.000 }
gfCNCPoint4[11223] = {X 163.3221, Y 17.4615, Z -5.5000, A 0.000, B 0.000, C 0.000 }
gfCNCPoint4[11224] = {X 163.2218, Y 18.3516, Z -5.5000, A 0.000, B 0.000, C 0.000 }
gfCNCPoint4[11225] = {X 162.9260, Y 19.1971, Z -5.5000, A 0.000, B 0.000, C 0.000 }
gfCNCPoint4[11226] = {X 162.4494, Y 19.9555, Z -5.5000, A 0.000, B 0.000, C 0.000 }
gfCNCPoint4[11227] = {X 161.8160, Y 20.5889, Z -5.5000, A 0.000, B 0.000, C 0.000 }
gfCNCPoint4[11228] = {X 161.0576, Y 21.0654, Z -5.5000, A 0.000, B 0.000, C 0.000 }
gfCNCPoint4[11229] = {X 160.2122, Y 21.3613, Z -5.5000, A 0.000, B 0.000, C 0.000 }
gfCNCPoint4[11230] = {X 159.3221, Y 21.4615, Z -5.5000, A 0.000, B 0.000, C 0.000 }
gfCNCPoint4[11231] = {X 158.6805, Y 21.4615, Z -5.5000, A 0.000, B 0.000, C 0.000 }
gfCNCPoint4[11232] = {X 157.8710, Y 21.3762, Z -5.5000, A 0.000, B 0.000, C 0.000 }
gfCNCPoint4[11233] = {X 157.0952, Y 21.1301, Z -5.5000, A 0.000, B 0.000, C 0.000 }
gfCNCPoint4[11234] = {X 156.3845, Y 20.7332, Z -5.5000, A 0.000, B 0.000, C 0.000 }
gfCNCPoint4[11235] = {X 155.7680, Y 20.2017, Z -5.5000, A 0.000, B 0.000, C 0.000 }
gfCNCPoint4[11236] = {X 155.2709, Y 19.5572, Z -5.5000, A 0.000, B 0.000, C 0.000 }
gfCNCPoint4[11237] = {X 151.9567, Y 19.5585, Z -5.5000, A 0.000, B 0.000, C 0.000 }
gfCNCPoint4[11238] = {X 151.9554, Y 40.9999, Z -5.5000, A 0.000, B 0.000, C 0.000 }
gfCNCPoint4[11239] = {X 152.5009, Y 41.5871, Z -5.5000, A 0.000, B 0.000, C 0.000 }
gfCNCPoint4[11240] = {X 152.5891, Y 41.6922, Z -5.5000, A 0.000, B 0.000, C 0.000 }
gfCNCPoint4[11241] = {X 153.0750, Y 42.4562, Z -5.5000, A 0.000, B 0.000, C 0.000 }
gfCNCPoint4[11242] = {X 153.3781, Y 43.3095, Z -5.5000, A 0.000, B 0.000, C 0.000 }
gfCNCPoint4[11243] = {X 153.4831, Y 44.2089, Z -5.5000, A 0.000, B 0.000, C 0.000 }
gfCNCPoint4[11244] = {X 153.4829, Y 45.0384, Z -5.5000, A 0.000, B 0.000, C 0.000 }
gfCNCPoint4[11245] = {X 153.3753, Y 45.9222, Z -5.5000, A 0.000, B 0.000, C 0.000 }
gfCNCPoint4[11246] = {X 153.0750, Y 46.7602, Z -5.5000, A 0.000, B 0.000, C 0.000 }
gfCNCPoint4[11247] = {X 152.5967, Y 47.5111, Z -5.5000, A 0.000, B 0.000, C 0.000 }
gfCNCPoint4[11248] = {X 151.9642, Y 48.1376, Z -5.5000, A 0.000, B 0.000, C 0.000 }
gfCNCPoint4[11249] = {X 151.2087, Y 48.6086, Z -5.5000, A 0.000, B 0.000, C 0.000 }
gfCNCPoint4[11250] = {X 150.3678, Y 48.9009, Z -5.5000, A 0.000, B 0.000, C 0.000 }
gfCNCPoint4[11251] = {X 149.4831, Y 49.0000, Z -5.5000, A 0.000, B 0.000, C 0.000 }
gfCNCPoint4[11252] = {X 143.0396, Y 49.0000, Z -5.5000, A 0.000, B 0.000, C 0.000 }
gfCNCPoint4[11253] = {X 142.1495, Y 48.8997, Z -5.5000, A 0.000, B 0.000, C 0.000 }
gfCNCPoint4[11254] = {X 141.3041, Y 48.6039, Z -5.5000, A 0.000, B 0.000, C 0.000 }
gfCNCPoint4[11255] = {X 140.5457, Y 48.1273, Z -5.5000, A 0.000, B 0.000, C 0.000 }
gfCNCPoint4[11256] = {X 139.9123, Y 47.4939, Z -5.5000, A 0.000, B 0.000, C 0.000 }
gfCNCPoint4[11257] = {X 139.4357, Y 46.7355, Z -5.5000, A 0.000, B 0.000, C 0.000 }
gfCNCPoint4[11258] = {X 139.1399, Y 45.8901, Z -5.5000, A 0.000, B 0.000, C 0.000 }
gfCNCPoint4[11259] = {X 139.0396, Y 45.0000, Z -5.5000, A 0.000, B 0.000, C 0.000 }
gfCNCPoint4[11260] = {X 139.0400, Y 44.1538, Z -5.5000, A 0.000, B 0.000, C 0.000 }
gfCNCPoint4[11261] = {X 139.1506, Y 43.2730, Z -5.5000, A 0.000, B 0.000, C 0.000 }
gfCNCPoint4[11262] = {X 139.4528, Y 42.4382, Z -5.5000, A 0.000, B 0.000, C 0.000 }
gfCNCPoint4[11263] = {X 139.9317, Y 41.6907, Z -5.5000, A 0.000, B 0.000, C 0.000 }
gfCNCPoint4[11264] = {X 140.5636, Y 41.0672, Z -5.5000, A 0.000, B 0.000, C 0.000 }
gfCNCPoint4[11265] = {X 140.5636, Y 30.3967, Z -5.5000, A 0.000, B 0.000, C 0.000 }
gfCNCPoint4[11266] = {X 136.4836, Y 30.3967, Z -5.5000, A 0.000, B 0.000, C 0.000 }
gfCNCPoint4[11267] = {X 136.4836, Y 30.3967, Z -2.5000, A 0.000, B 0.000, C 0.000 }
gfCNCPoint4[11268] = {X 136.4836, Y 30.3967, Z 11.0000, A 0.000, B 0.000, C 0.000 }
gfCNCPoint4[11269] = {X 137.6634, Y 74.8924, Z 11.0000, A 0.000, B 0.000, C 0.000 }
gfCNCPoint4[11270] = {X 137.6634, Y 74.8924, Z -2.5000, A 0.000, B 0.000, C 0.000 }
gfCNCPoint4[11271] = {X 137.6634, Y 74.8924, Z -5.5000, A 0.000, B 0.000, C 0.000 }
gfCNCPoint4[11272] = {X 140.6801, Y 77.6395, Z -5.5000, A 0.000, B 0.000, C 0.000 }
gfCNCPoint4[11273] = {X 155.6323, Y 61.2199, Z -5.5000, A 0.000, B 0.000, C 0.000 }
gfCNCPoint4[11274] = {X 155.2773, Y 60.5142, Z -5.5000, A 0.000, B 0.000, C 0.000 }
gfCNCPoint4[11275] = {X 155.0568, Y 59.7557, Z -5.5000, A 0.000, B 0.000, C 0.000 }
gfCNCPoint4[11276] = {X 154.9781, Y 58.9697, Z -5.5000, A 0.000, B 0.000, C 0.000 }
gfCNCPoint4[11277] = {X 154.9780, Y 58.0000, Z -5.5000, A 0.000, B 0.000, C 0.000 }
gfCNCPoint4[11278] = {X 155.0863, Y 57.0387, Z -5.5000, A 0.000, B 0.000, C 0.000 }
gfCNCPoint4[11279] = {X 155.4058, Y 56.1256, Z -5.5000, A 0.000, B 0.000, C 0.000 }
gfCNCPoint4[11280] = {X 155.9204, Y 55.3065, Z -5.5000, A 0.000, B 0.000, C 0.000 }
gfCNCPoint4[11281] = {X 156.6045, Y 54.6225, Z -5.5000, A 0.000, B 0.000, C 0.000 }
gfCNCPoint4[11282] = {X 157.4236, Y 54.1078, Z -5.5000, A 0.000, B 0.000, C 0.000 }
gfCNCPoint4[11283] = {X 158.3367, Y 53.7883, Z -5.5000, A 0.000, B 0.000, C 0.000 }
gfCNCPoint4[11284] = {X 159.2980, Y 53.6800, Z -5.5000, A 0.000, B 0.000, C 0.000 }
gfCNCPoint4[11285] = {X 178.5335, Y 53.6800, Z -5.5000, A 0.000, B 0.000, C 0.000 }
gfCNCPoint4[11286] = {X 179.4948, Y 53.7883, Z -5.5000, A 0.000, B 0.000, C 0.000 }
gfCNCPoint4[11287] = {X 180.4079, Y 54.1078, Z -5.5000, A 0.000, B 0.000, C 0.000 }
gfCNCPoint4[11288] = {X 181.2270, Y 54.6225, Z -5.5000, A 0.000, B 0.000, C 0.000 }
gfCNCPoint4[11289] = {X 181.9110, Y 55.3065, Z -5.5000, A 0.000, B 0.000, C 0.000 }
gfCNCPoint4[11290] = {X 182.4257, Y 56.1256, Z -5.5000, A 0.000, B 0.000, C 0.000 }
gfCNCPoint4[11291] = {X 182.7452, Y 57.0387, Z -5.5000, A 0.000, B 0.000, C 0.000 }
gfCNCPoint4[11292] = {X 182.8535, Y 58.0000, Z -5.5000, A 0.000, B 0.000, C 0.000 }
gfCNCPoint4[11293] = {X 182.8535, Y 58.9342, Z -5.5000, A 0.000, B 0.000, C 0.000 }
gfCNCPoint4[11294] = {X 182.7808, Y 59.7232, Z -5.5000, A 0.000, B 0.000, C 0.000 }
gfCNCPoint4[11295] = {X 182.5653, Y 60.4856, Z -5.5000, A 0.000, B 0.000, C 0.000 }
gfCNCPoint4[11296] = {X 182.2141, Y 61.1959, Z -5.5000, A 0.000, B 0.000, C 0.000 }
gfCNCPoint4[11297] = {X 209.4792, Y 90.9542, Z -5.5000, A 0.000, B 0.000, C 0.000 }
gfCNCPoint4[11298] = {X 210.1360, Y 91.6206, Z -5.5000, A 0.000, B 0.000, C 0.000 }
gfCNCPoint4[11299] = {X 210.8395, Y 92.2374, Z -5.5000, A 0.000, B 0.000, C 0.000 }
gfCNCPoint4[11300] = {X 211.1137, Y 92.4110, Z -5.5000, A 0.000, B 0.000, C 0.000 }
gfCNCPoint4[11301] = {X 211.4211, Y 92.5149, Z -5.5000, A 0.000, B 0.000, C 0.000 }
gfCNCPoint4[11302] = {X 213.4040, Y 92.8242, Z -5.5000, A 0.000, B 0.000, C 0.000 }
gfCNCPoint4[11303] = {X 214.4546, Y 92.7355, Z -5.5000, A 0.000, B 0.000, C 0.000 }
gfCNCPoint4[11304] = {X 215.5073, Y 92.6752, Z -5.5000, A 0.000, B 0.000, C 0.000 }
gfCNCPoint4[11305] = {X 216.1773, Y 92.6021, Z -5.5000, A 0.000, B 0.000, C 0.000 }
gfCNCPoint4[11306] = {X 216.8226, Y 92.4071, Z -5.5000, A 0.000, B 0.000, C 0.000 }
gfCNCPoint4[11307] = {X 217.4210, Y 92.0967, Z -5.5000, A 0.000, B 0.000, C 0.000 }
gfCNCPoint4[11308] = {X 222.9613, Y 88.5213, Z -5.5000, A 0.000, B 0.000, C 0.000 }
gfCNCPoint4[11309] = {X 245.8278, Y 73.8996, Z -5.5000, A 0.000, B 0.000, C 0.000 }
gfCNCPoint4[11310] = {X 221.6305, Y 64.4041, Z -5.5000, A 0.000, B 0.000, C 0.000 }
gfCNCPoint4[11311] = {X 219.8632, Y 63.8125, Z -5.5000, A 0.000, B 0.000, C 0.000 }
gfCNCPoint4[11312] = {X 218.0398, Y 63.4266, Z -5.5000, A 0.000, B 0.000, C 0.000 }
gfCNCPoint4[11313] = {X 216.1843, Y 63.2516, Z -5.5000, A 0.000, B 0.000, C 0.000 }
gfCNCPoint4[11314] = {X 215.2524, Y 63.1173, Z -5.5000, A 0.000, B 0.000, C 0.000 }
gfCNCPoint4[11315] = {X 214.3718, Y 62.7843, Z -5.5000, A 0.000, B 0.000, C 0.000 }
gfCNCPoint4[11316] = {X 213.5842, Y 62.2685, Z -5.5000, A 0.000, B 0.000, C 0.000 }
gfCNCPoint4[11317] = {X 212.9270, Y 61.5942, Z -5.5000, A 0.000, B 0.000, C 0.000 }
gfCNCPoint4[11318] = {X 212.4315, Y 60.7937, Z -5.5000, A 0.000, B 0.000, C 0.000 }
gfCNCPoint4[11319] = {X 212.1213, Y 59.9048, Z -5.5000, A 0.000, B 0.000, C 0.000 }
gfCNCPoint4[11320] = {X 212.0110, Y 58.9697, Z -5.5000, A 0.000, B 0.000, C 0.000 }
gfCNCPoint4[11321] = {X 212.0108, Y 58.0000, Z -5.5000, A 0.000, B 0.000, C 0.000 }
gfCNCPoint4[11322] = {X 212.1191, Y 57.0387, Z -5.5000, A 0.000, B 0.000, C 0.000 }
gfCNCPoint4[11323] = {X 212.4386, Y 56.1256, Z -5.5000, A 0.000, B 0.000, C 0.000 }
gfCNCPoint4[11324] = {X 212.9533, Y 55.3065, Z -5.5000, A 0.000, B 0.000, C 0.000 }
gfCNCPoint4[11325] = {X 213.6373, Y 54.6225, Z -5.5000, A 0.000, B 0.000, C 0.000 }
gfCNCPoint4[11326] = {X 214.4564, Y 54.1078, Z -5.5000, A 0.000, B 0.000, C 0.000 }
gfCNCPoint4[11327] = {X 215.3695, Y 53.7883, Z -5.5000, A 0.000, B 0.000, C 0.000 }
gfCNCPoint4[11328] = {X 216.3308, Y 53.6800, Z -5.5000, A 0.000, B 0.000, C 0.000 }
gfCNCPoint4[11329] = {X 237.2617, Y 53.6800, Z -5.5000, A 0.000, B 0.000, C 0.000 }
gfCNCPoint4[11330] = {X 238.2230, Y 53.7883, Z -5.5000, A 0.000, B 0.000, C 0.000 }
gfCNCPoint4[11331] = {X 239.1361, Y 54.1078, Z -5.5000, A 0.000, B 0.000, C 0.000 }
gfCNCPoint4[11332] = {X 239.9552, Y 54.6225, Z -5.5000, A 0.000, B 0.000, C 0.000 }
gfCNCPoint4[11333] = {X 240.6392, Y 55.3065, Z -5.5000, A 0.000, B 0.000, C 0.000 }
gfCNCPoint4[11334] = {X 241.1539, Y 56.1256, Z -5.5000, A 0.000, B 0.000, C 0.000 }
gfCNCPoint4[11335] = {X 241.4734, Y 57.0387, Z -5.5000, A 0.000, B 0.000, C 0.000 }
gfCNCPoint4[11336] = {X 241.5817, Y 58.0000, Z -5.5000, A 0.000, B 0.000, C 0.000 }
gfCNCPoint4[11337] = {X 241.5817, Y 58.2321, Z -5.5000, A 0.000, B 0.000, C 0.000 }
gfCNCPoint4[11338] = {X 248.1142, Y 60.7793, Z -5.5000, A 0.000, B 0.000, C 0.000 }
gfCNCPoint4[11339] = {X 275.6325, Y 71.7019, Z -5.5000, A 0.000, B 0.000, C 0.000 }
gfCNCPoint4[11340] = {X 275.6338, Y 63.2124, Z -5.5000, A 0.000, B 0.000, C 0.000 }
gfCNCPoint4[11341] = {X 274.7821, Y 63.0032, Z -5.5000, A 0.000, B 0.000, C 0.000 }
gfCNCPoint4[11342] = {X 273.9902, Y 62.6265, Z -5.5000, A 0.000, B 0.000, C 0.000 }
gfCNCPoint4[11343] = {X 273.2907, Y 62.0975, Z -5.5000, A 0.000, B 0.000, C 0.000 }
gfCNCPoint4[11344] = {X 272.7125, Y 61.4382, Z -5.5000, A 0.000, B 0.000, C 0.000 }
gfCNCPoint4[11345] = {X 272.2793, Y 60.6757, Z -5.5000, A 0.000, B 0.000, C 0.000 }
gfCNCPoint4[11346] = {X 272.0091, Y 59.8414, Z -5.5000, A 0.000, B 0.000, C 0.000 }
gfCNCPoint4[11347] = {X 271.9128, Y 58.9697, Z -5.5000, A 0.000, B 0.000, C 0.000 }
gfCNCPoint4[11348] = {X 271.9127, Y 58.0000, Z -5.5000, A 0.000, B 0.000, C 0.000 }
gfCNCPoint4[11349] = {X 272.0210, Y 57.0387, Z -5.5000, A 0.000, B 0.000, C 0.000 }
gfCNCPoint4[11350] = {X 272.3405, Y 56.1256, Z -5.5000, A 0.000, B 0.000, C 0.000 }
gfCNCPoint4[11351] = {X 272.8552, Y 55.3065, Z -5.5000, A 0.000, B 0.000, C 0.000 }
gfCNCPoint4[11352] = {X 273.5392, Y 54.6225, Z -5.5000, A 0.000, B 0.000, C 0.000 }
gfCNCPoint4[11353] = {X 274.3583, Y 54.1078, Z -5.5000, A 0.000, B 0.000, C 0.000 }
gfCNCPoint4[11354] = {X 275.2714, Y 53.7883, Z -5.5000, A 0.000, B 0.000, C 0.000 }
gfCNCPoint4[11355] = {X 276.2327, Y 53.6800, Z -5.5000, A 0.000, B 0.000, C 0.000 }
gfCNCPoint4[11356] = {X 292.7731, Y 53.6800, Z -5.5000, A 0.000, B 0.000, C 0.000 }
gfCNCPoint4[11357] = {X 293.7344, Y 53.7883, Z -5.5000, A 0.000, B 0.000, C 0.000 }
gfCNCPoint4[11358] = {X 294.6475, Y 54.1078, Z -5.5000, A 0.000, B 0.000, C 0.000 }
gfCNCPoint4[11359] = {X 295.4666, Y 54.6225, Z -5.5000, A 0.000, B 0.000, C 0.000 }
gfCNCPoint4[11360] = {X 296.1506, Y 55.3065, Z -5.5000, A 0.000, B 0.000, C 0.000 }
gfCNCPoint4[11361] = {X 296.6653, Y 56.1256, Z -5.5000, A 0.000, B 0.000, C 0.000 }
gfCNCPoint4[11362] = {X 296.9848, Y 57.0387, Z -5.5000, A 0.000, B 0.000, C 0.000 }
gfCNCPoint4[11363] = {X 297.0931, Y 58.0000, Z -5.5000, A 0.000, B 0.000, C 0.000 }
gfCNCPoint4[11364] = {X 297.0931, Y 58.9351, Z -5.5000, A 0.000, B 0.000, C 0.000 }
gfCNCPoint4[11365] = {X 297.0009, Y 59.8116, Z -5.5000, A 0.000, B 0.000, C 0.000 }
gfCNCPoint4[11366] = {X 296.7334, Y 60.6513, Z -5.5000, A 0.000, B 0.000, C 0.000 }
gfCNCPoint4[11367] = {X 296.3016, Y 61.4197, Z -5.5000, A 0.000, B 0.000, C 0.000 }
gfCNCPoint4[11368] = {X 295.7234, Y 62.0848, Z -5.5000, A 0.000, B 0.000, C 0.000 }
gfCNCPoint4[11369] = {X 295.0226, Y 62.6193, Z -5.5000, A 0.000, B 0.000, C 0.000 }
gfCNCPoint4[11370] = {X 294.2283, Y 63.0011, Z -5.5000, A 0.000, B 0.000, C 0.000 }
gfCNCPoint4[11371] = {X 293.3731, Y 63.2144, Z -5.5000, A 0.000, B 0.000, C 0.000 }
gfCNCPoint4[11372] = {X 293.3846, Y 92.7808, Z -5.5000, A 0.000, B 0.000, C 0.000 }
gfCNCPoint4[11373] = {X 294.2372, Y 92.9983, Z -5.5000, A 0.000, B 0.000, C 0.000 }
gfCNCPoint4[11374] = {X 295.0286, Y 93.3828, Z -5.5000, A 0.000, B 0.000, C 0.000 }
gfCNCPoint4[11375] = {X 295.7265, Y 93.9186, Z -5.5000, A 0.000, B 0.000, C 0.000 }
gfCNCPoint4[11376] = {X 296.3024, Y 94.5838, Z -5.5000, A 0.000, B 0.000, C 0.000 }
gfCNCPoint4[11377] = {X 296.7327, Y 95.3513, Z -5.5000, A 0.000, B 0.000, C 0.000 }
gfCNCPoint4[11378] = {X 296.9999, Y 96.1896, Z -5.5000, A 0.000, B 0.000, C 0.000 }
gfCNCPoint4[11379] = {X 297.0931, Y 97.0645, Z -5.5000, A 0.000, B 0.000, C 0.000 }
gfCNCPoint4[11380] = {X 297.0931, Y 98.0000, Z -5.5000, A 0.000, B 0.000, C 0.000 }
gfCNCPoint4[11381] = {X 296.9848, Y 98.9613, Z -5.5000, A 0.000, B 0.000, C 0.000 }
gfCNCPoint4[11382] = {X 296.6653, Y 99.8744, Z -5.5000, A 0.000, B 0.000, C 0.000 }
gfCNCPoint4[11383] = {X 296.1506, Y 100.6935, Z -5.5000, A 0.000, B 0.000, C 0.000 }
gfCNCPoint4[11384] = {X 295.4666, Y 101.3775, Z -5.5000, A 0.000, B 0.000, C 0.000 }
gfCNCPoint4[11385] = {X 294.6475, Y 101.8922, Z -5.5000, A 0.000, B 0.000, C 0.000 }
gfCNCPoint4[11386] = {X 293.7344, Y 102.2117, Z -5.5000, A 0.000, B 0.000, C 0.000 }
gfCNCPoint4[11387] = {X 292.7731, Y 102.3200, Z -5.5000, A 0.000, B 0.000, C 0.000 }
gfCNCPoint4[11388] = {X 276.2327, Y 102.3200, Z -5.5000, A 0.000, B 0.000, C 0.000 }
gfCNCPoint4[11389] = {X 275.2714, Y 102.2117, Z -5.5000, A 0.000, B 0.000, C 0.000 }
gfCNCPoint4[11390] = {X 274.3583, Y 101.8922, Z -5.5000, A 0.000, B 0.000, C 0.000 }
gfCNCPoint4[11391] = {X 273.5392, Y 101.3775, Z -5.5000, A 0.000, B 0.000, C 0.000 }
gfCNCPoint4[11392] = {X 272.8552, Y 100.6935, Z -5.5000, A 0.000, B 0.000, C 0.000 }
gfCNCPoint4[11393] = {X 272.3405, Y 99.8744, Z -5.5000, A 0.000, B 0.000, C 0.000 }
gfCNCPoint4[11394] = {X 272.0210, Y 98.9613, Z -5.5000, A 0.000, B 0.000, C 0.000 }
gfCNCPoint4[11395] = {X 271.9127, Y 98.0000, Z -5.5000, A 0.000, B 0.000, C 0.000 }
gfCNCPoint4[11396] = {X 271.9127, Y 97.0659, Z -5.5000, A 0.000, B 0.000, C 0.000 }
gfCNCPoint4[11397] = {X 272.0026, Y 96.1891, Z -5.5000, A 0.000, B 0.000, C 0.000 }
gfCNCPoint4[11398] = {X 272.2686, Y 95.3488, Z -5.5000, A 0.000, B 0.000, C 0.000 }
gfCNCPoint4[11399] = {X 272.6996, Y 94.5800, Z -5.5000, A 0.000, B 0.000, C 0.000 }
gfCNCPoint4[11400] = {X 273.2777, Y 93.9146, Z -5.5000, A 0.000, B 0.000, C 0.000 }
gfCNCPoint4[11401] = {X 273.9788, Y 93.3805, Z -5.5000, A 0.000, B 0.000, C 0.000 }
gfCNCPoint4[11402] = {X 274.7737, Y 92.9997, Z -5.5000, A 0.000, B 0.000, C 0.000 }
gfCNCPoint4[11403] = {X 275.6294, Y 92.7883, Z -5.5000, A 0.000, B 0.000, C 0.000 }
gfCNCPoint4[11404] = {X 275.6294, Y 85.5950, Z -5.5000, A 0.000, B 0.000, C 0.000 }
gfCNCPoint4[11405] = {X 262.6397, Y 80.5030, Z -5.5000, A 0.000, B 0.000, C 0.000 }
gfCNCPoint4[11406] = {X 262.2775, Y 80.7316, Z -5.5000, A 0.000, B 0.000, C 0.000 }
gfCNCPoint4[11407] = {X 237.7969, Y 96.5882, Z -5.5000, A 0.000, B 0.000, C 0.000 }
gfCNCPoint4[11408] = {X 237.7998, Y 97.0649, Z -5.5000, A 0.000, B 0.000, C 0.000 }
gfCNCPoint4[11409] = {X 237.7998, Y 98.0000, Z -5.5000, A 0.000, B 0.000, C 0.000 }
gfCNCPoint4[11410] = {X 237.6915, Y 98.9613, Z -5.5000, A 0.000, B 0.000, C 0.000 }
gfCNCPoint4[11411] = {X 237.3720, Y 99.8744, Z -5.5000, A 0.000, B 0.000, C 0.000 }
gfCNCPoint4[11412] = {X 236.8573, Y 100.6935, Z -5.5000, A 0.000, B 0.000, C 0.000 }
gfCNCPoint4[11413] = {X 236.1733, Y 101.3775, Z -5.5000, A 0.000, B 0.000, C 0.000 }
gfCNCPoint4[11414] = {X 235.3542, Y 101.8922, Z -5.5000, A 0.000, B 0.000, C 0.000 }
gfCNCPoint4[11415] = {X 234.4411, Y 102.2117, Z -5.5000, A 0.000, B 0.000, C 0.000 }
gfCNCPoint4[11416] = {X 233.4798, Y 102.3200, Z -5.5000, A 0.000, B 0.000, C 0.000 }
gfCNCPoint4[11417] = {X 214.1790, Y 102.3200, Z -5.5000, A 0.000, B 0.000, C 0.000 }
gfCNCPoint4[11418] = {X 213.7862, Y 102.3021, Z -5.5000, A 0.000, B 0.000, C 0.000 }
gfCNCPoint4[11419] = {X 213.3966, Y 102.2485, Z -5.5000, A 0.000, B 0.000, C 0.000 }
gfCNCPoint4[11420] = {X 213.0070, Y 102.3021, Z -5.5000, A 0.000, B 0.000, C 0.000 }
gfCNCPoint4[11421] = {X 212.6141, Y 102.3200, Z -5.5000, A 0.000, B 0.000, C 0.000 }
gfCNCPoint4[11422] = {X 194.9870, Y 102.3200, Z -5.5000, A 0.000, B 0.000, C 0.000 }
gfCNCPoint4[11423] = {X 194.0257, Y 102.2117, Z -5.5000, A 0.000, B 0.000, C 0.000 }
gfCNCPoint4[11424] = {X 193.1126, Y 101.8922, Z -5.5000, A 0.000, B 0.000, C 0.000 }
gfCNCPoint4[11425] = {X 192.2935, Y 101.3775, Z -5.5000, A 0.000, B 0.000, C 0.000 }
gfCNCPoint4[11426] = {X 191.6094, Y 100.6935, Z -5.5000, A 0.000, B 0.000, C 0.000 }
gfCNCPoint4[11427] = {X 191.0948, Y 99.8744, Z -5.5000, A 0.000, B 0.000, C 0.000 }
gfCNCPoint4[11428] = {X 190.7753, Y 98.9613, Z -5.5000, A 0.000, B 0.000, C 0.000 }
gfCNCPoint4[11429] = {X 190.6670, Y 98.0000, Z -5.5000, A 0.000, B 0.000, C 0.000 }
gfCNCPoint4[11430] = {X 190.6670, Y 97.0659, Z -5.5000, A 0.000, B 0.000, C 0.000 }
gfCNCPoint4[11431] = {X 190.7727, Y 96.1162, Z -5.5000, A 0.000, B 0.000, C 0.000 }
gfCNCPoint4[11432] = {X 191.0846, Y 95.2129, Z -5.5000, A 0.000, B 0.000, C 0.000 }
gfCNCPoint4[11433] = {X 191.5874, Y 94.4003, Z -5.5000, A 0.000, B 0.000, C 0.000 }
gfCNCPoint4[11434] = {X 188.5647, Y 91.1002, Z -5.5000, A 0.000, B 0.000, C 0.000 }
gfCNCPoint4[11435] = {X 150.0898, Y 91.1002, Z -5.5000, A 0.000, B 0.000, C 0.000 }
gfCNCPoint4[11436] = {X 147.1452, Y 94.3626, Z -5.5000, A 0.000, B 0.000, C 0.000 }
gfCNCPoint4[11437] = {X 147.6640, Y 95.1839, Z -5.5000, A 0.000, B 0.000, C 0.000 }
gfCNCPoint4[11438] = {X 147.9873, Y 96.1000, Z -5.5000, A 0.000, B 0.000, C 0.000 }
gfCNCPoint4[11439] = {X 148.0991, Y 97.0650, Z -5.5000, A 0.000, B 0.000, C 0.000 }
gfCNCPoint4[11440] = {X 148.0991, Y 98.0000, Z -5.5000, A 0.000, B 0.000, C 0.000 }
gfCNCPoint4[11441] = {X 147.9908, Y 98.9613, Z -5.5000, A 0.000, B 0.000, C 0.000 }
gfCNCPoint4[11442] = {X 147.6713, Y 99.8744, Z -5.5000, A 0.000, B 0.000, C 0.000 }
gfCNCPoint4[11443] = {X 147.1566, Y 100.6935, Z -5.5000, A 0.000, B 0.000, C 0.000 }
gfCNCPoint4[11444] = {X 146.4726, Y 101.3775, Z -5.5000, A 0.000, B 0.000, C 0.000 }
gfCNCPoint4[11445] = {X 145.6535, Y 101.8922, Z -5.5000, A 0.000, B 0.000, C 0.000 }
gfCNCPoint4[11446] = {X 144.7404, Y 102.2117, Z -5.5000, A 0.000, B 0.000, C 0.000 }
gfCNCPoint4[11447] = {X 143.7791, Y 102.3200, Z -5.5000, A 0.000, B 0.000, C 0.000 }
gfCNCPoint4[11448] = {X 125.0000, Y 102.3200, Z -5.5000, A 0.000, B 0.000, C 0.000 }
gfCNCPoint4[11449] = {X 124.0387, Y 102.2117, Z -5.5000, A 0.000, B 0.000, C 0.000 }
gfCNCPoint4[11450] = {X 123.1256, Y 101.8922, Z -5.5000, A 0.000, B 0.000, C 0.000 }
gfCNCPoint4[11451] = {X 122.3065, Y 101.3775, Z -5.5000, A 0.000, B 0.000, C 0.000 }
gfCNCPoint4[11452] = {X 121.6225, Y 100.6935, Z -5.5000, A 0.000, B 0.000, C 0.000 }
gfCNCPoint4[11453] = {X 121.1078, Y 99.8744, Z -5.5000, A 0.000, B 0.000, C 0.000 }
gfCNCPoint4[11454] = {X 120.7883, Y 98.9613, Z -5.5000, A 0.000, B 0.000, C 0.000 }
gfCNCPoint4[11455] = {X 120.6800, Y 98.0000, Z -5.5000, A 0.000, B 0.000, C 0.000 }
gfCNCPoint4[11456] = {X 120.6800, Y 97.0659, Z -5.5000, A 0.000, B 0.000, C 0.000 }
gfCNCPoint4[11457] = {X 120.7832, Y 96.1274, Z -5.5000, A 0.000, B 0.000, C 0.000 }
gfCNCPoint4[11458] = {X 121.0878, Y 95.2338, Z -5.5000, A 0.000, B 0.000, C 0.000 }
gfCNCPoint4[11459] = {X 121.5792, Y 94.4276, Z -5.5000, A 0.000, B 0.000, C 0.000 }
gfCNCPoint4[11460] = {X 122.2341, Y 93.7475, Z -5.5000, A 0.000, B 0.000, C 0.000 }
gfCNCPoint4[11461] = {X 123.0211, Y 93.2258, Z -5.5000, A 0.000, B 0.000, C 0.000 }
gfCNCPoint4[11462] = {X 123.9026, Y 92.8876, Z -5.5000, A 0.000, B 0.000, C 0.000 }
gfCNCPoint4[11463] = {X 124.8365, Y 92.7490, Z -5.5000, A 0.000, B 0.000, C 0.000 }
gfCNCPoint4[11464] = {X 124.8811, Y 92.7317, Z -5.5000, A 0.000, B 0.000, C 0.000 }
gfCNCPoint4[11465] = {X 124.9278, Y 92.7211, Z -5.5000, A 0.000, B 0.000, C 0.000 }
gfCNCPoint4[11466] = {X 125.4494, Y 92.6438, Z -5.5000, A 0.000, B 0.000, C 0.000 }
gfCNCPoint4[11467] = {X 126.2805, Y 92.5039, Z -5.5000, A 0.000, B 0.000, C 0.000 }
gfCNCPoint4[11468] = {X 127.1000, Y 92.3075, Z -5.5000, A 0.000, B 0.000, C 0.000 }
gfCNCPoint4[11469] = {X 128.3215, Y 91.1563, Z -5.5000, A 0.000, B 0.000, C 0.000 }
gfCNCPoint4[11470] = {X 129.4786, Y 89.9402, Z -5.5000, A 0.000, B 0.000, C 0.000 }
gfCNCPoint4[11471] = {X 140.6801, Y 77.6395, Z -5.5000, A 0.000, B 0.000, C 0.000 }
gfCNCPoint4[11472] = {X 137.7226, Y 74.9463, Z -5.5000, A 0.000, B 0.000, C 0.000 }
gfCNCPoint4[11473] = {X 140.7392, Y 77.6933, Z -5.5000, A 0.000, B 0.000, C 0.000 }
gfCNCPoint4[11474] = {X 155.7325, Y 61.2287, Z -5.5000, A 0.000, B 0.000, C 0.000 }
gfCNCPoint4[11475] = {X 155.3667, Y 60.5224, Z -5.5000, A 0.000, B 0.000, C 0.000 }
gfCNCPoint4[11476] = {X 155.1392, Y 59.7603, Z -5.5000, A 0.000, B 0.000, C 0.000 }
gfCNCPoint4[11477] = {X 155.0581, Y 58.9691, Z -5.5000, A 0.000, B 0.000, C 0.000 }
gfCNCPoint4[11478] = {X 155.0580, Y 58.0000, Z -5.5000, A 0.000, B 0.000, C 0.000 }
gfCNCPoint4[11479] = {X 155.1643, Y 57.0565, Z -5.5000, A 0.000, B 0.000, C 0.000 }
gfCNCPoint4[11480] = {X 155.4778, Y 56.1603, Z -5.5000, A 0.000, B 0.000, C 0.000 }
gfCNCPoint4[11481] = {X 155.9830, Y 55.3564, Z -5.5000, A 0.000, B 0.000, C 0.000 }
gfCNCPoint4[11482] = {X 156.6544, Y 54.6850, Z -5.5000, A 0.000, B 0.000, C 0.000 }
gfCNCPoint4[11483] = {X 157.4583, Y 54.1799, Z -5.5000, A 0.000, B 0.000, C 0.000 }
gfCNCPoint4[11484] = {X 158.3545, Y 53.8663, Z -5.5000, A 0.000, B 0.000, C 0.000 }
gfCNCPoint4[11485] = {X 159.2980, Y 53.7600, Z -5.5000, A 0.000, B 0.000, C 0.000 }
gfCNCPoint4[11486] = {X 178.5335, Y 53.7600, Z -5.5000, A 0.000, B 0.000, C 0.000 }
gfCNCPoint4[11487] = {X 179.4770, Y 53.8663, Z -5.5000, A 0.000, B 0.000, C 0.000 }
gfCNCPoint4[11488] = {X 180.3732, Y 54.1799, Z -5.5000, A 0.000, B 0.000, C 0.000 }
gfCNCPoint4[11489] = {X 181.1771, Y 54.6850, Z -5.5000, A 0.000, B 0.000, C 0.000 }
gfCNCPoint4[11490] = {X 181.8485, Y 55.3564, Z -5.5000, A 0.000, B 0.000, C 0.000 }
gfCNCPoint4[11491] = {X 182.3536, Y 56.1603, Z -5.5000, A 0.000, B 0.000, C 0.000 }
gfCNCPoint4[11492] = {X 182.6672, Y 57.0565, Z -5.5000, A 0.000, B 0.000, C 0.000 }
gfCNCPoint4[11493] = {X 182.7735, Y 58.0000, Z -5.5000, A 0.000, B 0.000, C 0.000 }
gfCNCPoint4[11494] = {X 182.7735, Y 58.9342, Z -5.5000, A 0.000, B 0.000, C 0.000 }
gfCNCPoint4[11495] = {X 182.6984, Y 59.7283, Z -5.5000, A 0.000, B 0.000, C 0.000 }
gfCNCPoint4[11496] = {X 182.4760, Y 60.4943, Z -5.5000, A 0.000, B 0.000, C 0.000 }
gfCNCPoint4[11497] = {X 182.1140, Y 61.2051, Z -5.5000, A 0.000, B 0.000, C 0.000 }
gfCNCPoint4[11498] = {X 209.4202, Y 91.0083, Z -5.5000, A 0.000, B 0.000, C 0.000 }
gfCNCPoint4[11499] = {X 210.0811, Y 91.6788, Z -5.5000, A 0.000, B 0.000, C 0.000 }
gfCNCPoint4[11500] = {X 210.7890, Y 92.2994, Z -5.5000, A 0.000, B 0.000, C 0.000 }
gfCNCPoint4[11501] = {X 211.0802, Y 92.4836, Z -5.5000, A 0.000, B 0.000, C 0.000 }
gfCNCPoint4[11502] = {X 211.4068, Y 92.5936, Z -5.5000, A 0.000, B 0.000, C 0.000 }
gfCNCPoint4[11503] = {X 213.4017, Y 92.9048, Z -5.5000, A 0.000, B 0.000, C 0.000 }
gfCNCPoint4[11504] = {X 214.4547, Y 92.8157, Z -5.5000, A 0.000, B 0.000, C 0.000 }
gfCNCPoint4[11505] = {X 215.5097, Y 92.7552, Z -5.5000, A 0.000, B 0.000, C 0.000 }
gfCNCPoint4[11506] = {X 216.1941, Y 92.6803, Z -5.5000, A 0.000, B 0.000, C 0.000 }
gfCNCPoint4[11507] = {X 216.8532, Y 92.4810, Z -5.5000, A 0.000, B 0.000, C 0.000 }
gfCNCPoint4[11508] = {X 217.4644, Y 92.1640, Z -5.5000, A 0.000, B 0.000, C 0.000 }
gfCNCPoint4[11509] = {X 223.0046, Y 88.5886, Z -5.5000, A 0.000, B 0.000, C 0.000 }
gfCNCPoint4[11510] = {X 246.0031, Y 73.8824, Z -5.5000, A 0.000, B 0.000, C 0.000 }
gfCNCPoint4[11511] = {X 221.6602, Y 64.3298, Z -5.5000, A 0.000, B 0.000, C 0.000 }
gfCNCPoint4[11512] = {X 219.8841, Y 63.7353, Z -5.5000, A 0.000, B 0.000, C 0.000 }
gfCNCPoint4[11513] = {X 218.0518, Y 63.3475, Z -5.5000, A 0.000, B 0.000, C 0.000 }
gfCNCPoint4[11514] = {X 216.1871, Y 63.1716, Z -5.5000, A 0.000, B 0.000, C 0.000 }
gfCNCPoint4[11515] = {X 215.2725, Y 63.0399, Z -5.5000, A 0.000, B 0.000, C 0.000 }
gfCNCPoint4[11516] = {X 214.4081, Y 62.7131, Z -5.5000, A 0.000, B 0.000, C 0.000 }
gfCNCPoint4[11517] = {X 213.6351, Y 62.2068, Z -5.5000, A 0.000, B 0.000, C 0.000 }
gfCNCPoint4[11518] = {X 212.9901, Y 61.5450, Z -5.5000, A 0.000, B 0.000, C 0.000 }
gfCNCPoint4[11519] = {X 212.5038, Y 60.7593, Z -5.5000, A 0.000, B 0.000, C 0.000 }
gfCNCPoint4[11520] = {X 212.1992, Y 59.8868, Z -5.5000, A 0.000, B 0.000, C 0.000 }
gfCNCPoint4[11521] = {X 212.0910, Y 58.9691, Z -5.5000, A 0.000, B 0.000, C 0.000 }
gfCNCPoint4[11522] = {X 212.0908, Y 58.0000, Z -5.5000, A 0.000, B 0.000, C 0.000 }
gfCNCPoint4[11523] = {X 212.1971, Y 57.0565, Z -5.5000, A 0.000, B 0.000, C 0.000 }
gfCNCPoint4[11524] = {X 212.5107, Y 56.1603, Z -5.5000, A 0.000, B 0.000, C 0.000 }
gfCNCPoint4[11525] = {X 213.0158, Y 55.3564, Z -5.5000, A 0.000, B 0.000, C 0.000 }
gfCNCPoint4[11526] = {X 213.6872, Y 54.6850, Z -5.5000, A 0.000, B 0.000, C 0.000 }
gfCNCPoint4[11527] = {X 214.4911, Y 54.1799, Z -5.5000, A 0.000, B 0.000, C 0.000 }
gfCNCPoint4[11528] = {X 215.3873, Y 53.8663, Z -5.5000, A 0.000, B 0.000, C 0.000 }
gfCNCPoint4[11529] = {X 216.3308, Y 53.7600, Z -5.5000, A 0.000, B 0.000, C 0.000 }
gfCNCPoint4[11530] = {X 237.2617, Y 53.7600, Z -5.5000, A 0.000, B 0.000, C 0.000 }
gfCNCPoint4[11531] = {X 238.2052, Y 53.8663, Z -5.5000, A 0.000, B 0.000, C 0.000 }
gfCNCPoint4[11532] = {X 239.1014, Y 54.1799, Z -5.5000, A 0.000, B 0.000, C 0.000 }
gfCNCPoint4[11533] = {X 239.9053, Y 54.6850, Z -5.5000, A 0.000, B 0.000, C 0.000 }
gfCNCPoint4[11534] = {X 240.5767, Y 55.3564, Z -5.5000, A 0.000, B 0.000, C 0.000 }
gfCNCPoint4[11535] = {X 241.0818, Y 56.1603, Z -5.5000, A 0.000, B 0.000, C 0.000 }
gfCNCPoint4[11536] = {X 241.3954, Y 57.0565, Z -5.5000, A 0.000, B 0.000, C 0.000 }
gfCNCPoint4[11537] = {X 241.5017, Y 58.0000, Z -5.5000, A 0.000, B 0.000, C 0.000 }
gfCNCPoint4[11538] = {X 241.5017, Y 58.2868, Z -5.5000, A 0.000, B 0.000, C 0.000 }
gfCNCPoint4[11539] = {X 248.0849, Y 60.8537, Z -5.5000, A 0.000, B 0.000, C 0.000 }
gfCNCPoint4[11540] = {X 275.7125, Y 71.8197, Z -5.5000, A 0.000, B 0.000, C 0.000 }
gfCNCPoint4[11541] = {X 275.7138, Y 63.1422, Z -5.5000, A 0.000, B 0.000, C 0.000 }
gfCNCPoint4[11542] = {X 274.8652, Y 62.9475, Z -5.5000, A 0.000, B 0.000, C 0.000 }
gfCNCPoint4[11543] = {X 274.0743, Y 62.5836, Z -5.5000, A 0.000, B 0.000, C 0.000 }
gfCNCPoint4[11544] = {X 273.3744, Y 62.0658, Z -5.5000, A 0.000, B 0.000, C 0.000 }
gfCNCPoint4[11545] = {X 272.7950, Y 61.4160, Z -5.5000, A 0.000, B 0.000, C 0.000 }
gfCNCPoint4[11546] = {X 272.3606, Y 60.6616, Z -5.5000, A 0.000, B 0.000, C 0.000 }
gfCNCPoint4[11547] = {X 272.0894, Y 59.8343, Z -5.5000, A 0.000, B 0.000, C 0.000 }
gfCNCPoint4[11548] = {X 271.9928, Y 58.9691, Z -5.5000, A 0.000, B 0.000, C 0.000 }
gfCNCPoint4[11549] = {X 271.9927, Y 58.0000, Z -5.5000, A 0.000, B 0.000, C 0.000 }
gfCNCPoint4[11550] = {X 272.0990, Y 57.0565, Z -5.5000, A 0.000, B 0.000, C 0.000 }
gfCNCPoint4[11551] = {X 272.4126, Y 56.1603, Z -5.5000, A 0.000, B 0.000, C 0.000 }
gfCNCPoint4[11552] = {X 272.9177, Y 55.3564, Z -5.5000, A 0.000, B 0.000, C 0.000 }
gfCNCPoint4[11553] = {X 273.5891, Y 54.6850, Z -5.5000, A 0.000, B 0.000, C 0.000 }
gfCNCPoint4[11554] = {X 274.3930, Y 54.1799, Z -5.5000, A 0.000, B 0.000, C 0.000 }
gfCNCPoint4[11555] = {X 275.2892, Y 53.8663, Z -5.5000, A 0.000, B 0.000, C 0.000 }
gfCNCPoint4[11556] = {X 276.2327, Y 53.7600, Z -5.5000, A 0.000, B 0.000, C 0.000 }
gfCNCPoint4[11557] = {X 292.7731, Y 53.7600, Z -5.5000, A 0.000, B 0.000, C 0.000 }
gfCNCPoint4[11558] = {X 293.7166, Y 53.8663, Z -5.5000, A 0.000, B 0.000, C 0.000 }
gfCNCPoint4[11559] = {X 294.6128, Y 54.1799, Z -5.5000, A 0.000, B 0.000, C 0.000 }
gfCNCPoint4[11560] = {X 295.4167, Y 54.6850, Z -5.5000, A 0.000, B 0.000, C 0.000 }
gfCNCPoint4[11561] = {X 296.0881, Y 55.3564, Z -5.5000, A 0.000, B 0.000, C 0.000 }
gfCNCPoint4[11562] = {X 296.5932, Y 56.1603, Z -5.5000, A 0.000, B 0.000, C 0.000 }
gfCNCPoint4[11563] = {X 296.9068, Y 57.0565, Z -5.5000, A 0.000, B 0.000, C 0.000 }
gfCNCPoint4[11564] = {X 297.0131, Y 58.0000, Z -5.5000, A 0.000, B 0.000, C 0.000 }
gfCNCPoint4[11565] = {X 297.0131, Y 58.9348, Z -5.5000, A 0.000, B 0.000, C 0.000 }
gfCNCPoint4[11566] = {X 296.9206, Y 59.8045, Z -5.5000, A 0.000, B 0.000, C 0.000 }
gfCNCPoint4[11567] = {X 296.6523, Y 60.6370, Z -5.5000, A 0.000, B 0.000, C 0.000 }
gfCNCPoint4[11568] = {X 296.2195, Y 61.3971, Z -5.5000, A 0.000, B 0.000, C 0.000 }
gfCNCPoint4[11569] = {X 295.6405, Y 62.0526, Z -5.5000, A 0.000, B 0.000, C 0.000 }
gfCNCPoint4[11570] = {X 294.9398, Y 62.5760, Z -5.5000, A 0.000, B 0.000, C 0.000 }
gfCNCPoint4[11571] = {X 294.1468, Y 62.9450, Z -5.5000, A 0.000, B 0.000, C 0.000 }
gfCNCPoint4[11572] = {X 293.2952, Y 63.1442, Z -5.5000, A 0.000, B 0.000, C 0.000 }
gfCNCPoint4[11573] = {X 293.3046, Y 92.8503, Z -5.5000, A 0.000, B 0.000, C 0.000 }
gfCNCPoint4[11574] = {X 294.1541, Y 93.0535, Z -5.5000, A 0.000, B 0.000, C 0.000 }
gfCNCPoint4[11575] = {X 294.9446, Y 93.4253, Z -5.5000, A 0.000, B 0.000, C 0.000 }
gfCNCPoint4[11576] = {X 295.6429, Y 93.9500, Z -5.5000, A 0.000, B 0.000, C 0.000 }
gfCNCPoint4[11577] = {X 296.2199, Y 94.6057, Z -5.5000, A 0.000, B 0.000, C 0.000 }
gfCNCPoint4[11578] = {X 296.6515, Y 95.3651, Z -5.5000, A 0.000, B 0.000, C 0.000 }
gfCNCPoint4[11579] = {X 296.9196, Y 96.1964, Z -5.5000, A 0.000, B 0.000, C 0.000 }
gfCNCPoint4[11580] = {X 297.0131, Y 97.0649, Z -5.5000, A 0.000, B 0.000, C 0.000 }
gfCNCPoint4[11581] = {X 297.0131, Y 98.0000, Z -5.5000, A 0.000, B 0.000, C 0.000 }
gfCNCPoint4[11582] = {X 296.9068, Y 98.9435, Z -5.5000, A 0.000, B 0.000, C 0.000 }
gfCNCPoint4[11583] = {X 296.5932, Y 99.8397, Z -5.5000, A 0.000, B 0.000, C 0.000 }
gfCNCPoint4[11584] = {X 296.0881, Y 100.6436, Z -5.5000, A 0.000, B 0.000, C 0.000 }
gfCNCPoint4[11585] = {X 295.4167, Y 101.3150, Z -5.5000, A 0.000, B 0.000, C 0.000 }
gfCNCPoint4[11586] = {X 294.6128, Y 101.8201, Z -5.5000, A 0.000, B 0.000, C 0.000 }
gfCNCPoint4[11587] = {X 293.7166, Y 102.1337, Z -5.5000, A 0.000, B 0.000, C 0.000 }
gfCNCPoint4[11588] = {X 292.7731, Y 102.2400, Z -5.5000, A 0.000, B 0.000, C 0.000 }
gfCNCPoint4[11589] = {X 276.2327, Y 102.2400, Z -5.5000, A 0.000, B 0.000, C 0.000 }
gfCNCPoint4[11590] = {X 275.2892, Y 102.1337, Z -5.5000, A 0.000, B 0.000, C 0.000 }
gfCNCPoint4[11591] = {X 274.3930, Y 101.8201, Z -5.5000, A 0.000, B 0.000, C 0.000 }
gfCNCPoint4[11592] = {X 273.5891, Y 101.3150, Z -5.5000, A 0.000, B 0.000, C 0.000 }
gfCNCPoint4[11593] = {X 272.9177, Y 100.6436, Z -5.5000, A 0.000, B 0.000, C 0.000 }
gfCNCPoint4[11594] = {X 272.4126, Y 99.8397, Z -5.5000, A 0.000, B 0.000, C 0.000 }
gfCNCPoint4[11595] = {X 272.0990, Y 98.9435, Z -5.5000, A 0.000, B 0.000, C 0.000 }
gfCNCPoint4[11596] = {X 271.9927, Y 98.0000, Z -5.5000, A 0.000, B 0.000, C 0.000 }
gfCNCPoint4[11597] = {X 271.9927, Y 97.0659, Z -5.5000, A 0.000, B 0.000, C 0.000 }
gfCNCPoint4[11598] = {X 272.0830, Y 96.1956, Z -5.5000, A 0.000, B 0.000, C 0.000 }
gfCNCPoint4[11599] = {X 272.3500, Y 95.3624, Z -5.5000, A 0.000, B 0.000, C 0.000 }
gfCNCPoint4[11600] = {X 272.7823, Y 94.6017, Z -5.5000, A 0.000, B 0.000, C 0.000 }
gfCNCPoint4[11601] = {X 273.3615, Y 93.9460, Z -5.5000, A 0.000, B 0.000, C 0.000 }
gfCNCPoint4[11602] = {X 274.0630, Y 93.4231, Z -5.5000, A 0.000, B 0.000, C 0.000 }
gfCNCPoint4[11603] = {X 274.8569, Y 93.0553, Z -5.5000, A 0.000, B 0.000, C 0.000 }
gfCNCPoint4[11604] = {X 275.7094, Y 92.8584, Z -5.5000, A 0.000, B 0.000, C 0.000 }
gfCNCPoint4[11605] = {X 275.7094, Y 85.5404, Z -5.5000, A 0.000, B 0.000, C 0.000 }
gfCNCPoint4[11606] = {X 262.6313, Y 80.4138, Z -5.5000, A 0.000, B 0.000, C 0.000 }
gfCNCPoint4[11607] = {X 262.2344, Y 80.6642, Z -5.5000, A 0.000, B 0.000, C 0.000 }
gfCNCPoint4[11608] = {X 237.7166, Y 96.5449, Z -5.5000, A 0.000, B 0.000, C 0.000 }
gfCNCPoint4[11609] = {X 237.7198, Y 97.0652, Z -5.5000, A 0.000, B 0.000, C 0.000 }
gfCNCPoint4[11610] = {X 237.7198, Y 98.0000, Z -5.5000, A 0.000, B 0.000, C 0.000 }
gfCNCPoint4[11611] = {X 237.6135, Y 98.9435, Z -5.5000, A 0.000, B 0.000, C 0.000 }
gfCNCPoint4[11612] = {X 237.2999, Y 99.8397, Z -5.5000, A 0.000, B 0.000, C 0.000 }
gfCNCPoint4[11613] = {X 236.7948, Y 100.6436, Z -5.5000, A 0.000, B 0.000, C 0.000 }
gfCNCPoint4[11614] = {X 236.1234, Y 101.3150, Z -5.5000, A 0.000, B 0.000, C 0.000 }
gfCNCPoint4[11615] = {X 235.3195, Y 101.8201, Z -5.5000, A 0.000, B 0.000, C 0.000 }
gfCNCPoint4[11616] = {X 234.4233, Y 102.1337, Z -5.5000, A 0.000, B 0.000, C 0.000 }
gfCNCPoint4[11617] = {X 233.4798, Y 102.2400, Z -5.5000, A 0.000, B 0.000, C 0.000 }
gfCNCPoint4[11618] = {X 214.1790, Y 102.2400, Z -5.5000, A 0.000, B 0.000, C 0.000 }
gfCNCPoint4[11619] = {X 213.7861, Y 102.2218, Z -5.5000, A 0.000, B 0.000, C 0.000 }
gfCNCPoint4[11620] = {X 213.3966, Y 102.1672, Z -5.5000, A 0.000, B 0.000, C 0.000 }
gfCNCPoint4[11621] = {X 213.0070, Y 102.2218, Z -5.5000, A 0.000, B 0.000, C 0.000 }
gfCNCPoint4[11622] = {X 212.6141, Y 102.2400, Z -5.5000, A 0.000, B 0.000, C 0.000 }
gfCNCPoint4[11623] = {X 194.9870, Y 102.2400, Z -5.5000, A 0.000, B 0.000, C 0.000 }
gfCNCPoint4[11624] = {X 194.0435, Y 102.1337, Z -5.5000, A 0.000, B 0.000, C 0.000 }
gfCNCPoint4[11625] = {X 193.1473, Y 101.8201, Z -5.5000, A 0.000, B 0.000, C 0.000 }
gfCNCPoint4[11626] = {X 192.3434, Y 101.3150, Z -5.5000, A 0.000, B 0.000, C 0.000 }
gfCNCPoint4[11627] = {X 191.6720, Y 100.6436, Z -5.5000, A 0.000, B 0.000, C 0.000 }
gfCNCPoint4[11628] = {X 191.1669, Y 99.8397, Z -5.5000, A 0.000, B 0.000, C 0.000 }
gfCNCPoint4[11629] = {X 190.8533, Y 98.9435, Z -5.5000, A 0.000, B 0.000, C 0.000 }
gfCNCPoint4[11630] = {X 190.7470, Y 98.0000, Z -5.5000, A 0.000, B 0.000, C 0.000 }
gfCNCPoint4[11631] = {X 190.7470, Y 97.0659, Z -5.5000, A 0.000, B 0.000, C 0.000 }
gfCNCPoint4[11632] = {X 190.8557, Y 96.1118, Z -5.5000, A 0.000, B 0.000, C 0.000 }
gfCNCPoint4[11633] = {X 191.1764, Y 95.2065, Z -5.5000, A 0.000, B 0.000, C 0.000 }
gfCNCPoint4[11634] = {X 191.6926, Y 94.3967, Z -5.5000, A 0.000, B 0.000, C 0.000 }
gfCNCPoint4[11635] = {X 188.5999, Y 91.0202, Z -5.5000, A 0.000, B 0.000, C 0.000 }
gfCNCPoint4[11636] = {X 150.0543, Y 91.0202, Z -5.5000, A 0.000, B 0.000, C 0.000 }
gfCNCPoint4[11637] = {X 147.0398, Y 94.3599, Z -5.5000, A 0.000, B 0.000, C 0.000 }
gfCNCPoint4[11638] = {X 147.5720, Y 95.1781, Z -5.5000, A 0.000, B 0.000, C 0.000 }
gfCNCPoint4[11639] = {X 147.9042, Y 96.0960, Z -5.5000, A 0.000, B 0.000, C 0.000 }
gfCNCPoint4[11640] = {X 148.0191, Y 97.0653, Z -5.5000, A 0.000, B 0.000, C 0.000 }
gfCNCPoint4[11641] = {X 148.0191, Y 98.0000, Z -5.5000, A 0.000, B 0.000, C 0.000 }
gfCNCPoint4[11642] = {X 147.9128, Y 98.9435, Z -5.5000, A 0.000, B 0.000, C 0.000 }
gfCNCPoint4[11643] = {X 147.5992, Y 99.8397, Z -5.5000, A 0.000, B 0.000, C 0.000 }
gfCNCPoint4[11644] = {X 147.0941, Y 100.6436, Z -5.5000, A 0.000, B 0.000, C 0.000 }
gfCNCPoint4[11645] = {X 146.4227, Y 101.3150, Z -5.5000, A 0.000, B 0.000, C 0.000 }
gfCNCPoint4[11646] = {X 145.6188, Y 101.8201, Z -5.5000, A 0.000, B 0.000, C 0.000 }
gfCNCPoint4[11647] = {X 144.7226, Y 102.1337, Z -5.5000, A 0.000, B 0.000, C 0.000 }
gfCNCPoint4[11648] = {X 143.7791, Y 102.2400, Z -5.5000, A 0.000, B 0.000, C 0.000 }
gfCNCPoint4[11649] = {X 125.0000, Y 102.2400, Z -5.5000, A 0.000, B 0.000, C 0.000 }
gfCNCPoint4[11650] = {X 124.0565, Y 102.1337, Z -5.5000, A 0.000, B 0.000, C 0.000 }
gfCNCPoint4[11651] = {X 123.1603, Y 101.8201, Z -5.5000, A 0.000, B 0.000, C 0.000 }
gfCNCPoint4[11652] = {X 122.3564, Y 101.3150, Z -5.5000, A 0.000, B 0.000, C 0.000 }
gfCNCPoint4[11653] = {X 121.6850, Y 100.6436, Z -5.5000, A 0.000, B 0.000, C 0.000 }
gfCNCPoint4[11654] = {X 121.1799, Y 99.8397, Z -5.5000, A 0.000, B 0.000, C 0.000 }
gfCNCPoint4[11655] = {X 120.8663, Y 98.9435, Z -5.5000, A 0.000, B 0.000, C 0.000 }
gfCNCPoint4[11656] = {X 120.7600, Y 98.0000, Z -5.5000, A 0.000, B 0.000, C 0.000 }
gfCNCPoint4[11657] = {X 120.7600, Y 97.0659, Z -5.5000, A 0.000, B 0.000, C 0.000 }
gfCNCPoint4[11658] = {X 120.8618, Y 96.1423, Z -5.5000, A 0.000, B 0.000, C 0.000 }
gfCNCPoint4[11659] = {X 121.1624, Y 95.2631, Z -5.5000, A 0.000, B 0.000, C 0.000 }
gfCNCPoint4[11660] = {X 121.6472, Y 94.4704, Z -5.5000, A 0.000, B 0.000, C 0.000 }
gfCNCPoint4[11661] = {X 122.2931, Y 93.8024, Z -5.5000, A 0.000, B 0.000, C 0.000 }
gfCNCPoint4[11662] = {X 123.0690, Y 93.2912, Z -5.5000, A 0.000, B 0.000, C 0.000 }
gfCNCPoint4[11663] = {X 123.9376, Y 92.9612, Z -5.5000, A 0.000, B 0.000, C 0.000 }
gfCNCPoint4[11664] = {X 124.8573, Y 92.8283, Z -5.5000, A 0.000, B 0.000, C 0.000 }
gfCNCPoint4[11665] = {X 124.8971, Y 92.8105, Z -5.5000, A 0.000, B 0.000, C 0.000 }
gfCNCPoint4[11666] = {X 124.9395, Y 92.8003, Z -5.5000, A 0.000, B 0.000, C 0.000 }
gfCNCPoint4[11667] = {X 125.4606, Y 92.7230, Z -5.5000, A 0.000, B 0.000, C 0.000 }
gfCNCPoint4[11668] = {X 126.3059, Y 92.5804, Z -5.5000, A 0.000, B 0.000, C 0.000 }
gfCNCPoint4[11669] = {X 127.1393, Y 92.3796, Z -5.5000, A 0.000, B 0.000, C 0.000 }
gfCNCPoint4[11670] = {X 128.3713, Y 91.2196, Z -5.5000, A 0.000, B 0.000, C 0.000 }
gfCNCPoint4[11671] = {X 129.5380, Y 89.9938, Z -5.5000, A 0.000, B 0.000, C 0.000 }
gfCNCPoint4[11672] = {X 140.7392, Y 77.6933, Z -5.5000, A 0.000, B 0.000, C 0.000 }
gfCNCPoint4[11673] = {X 137.7817, Y 75.0001, Z -5.5000, A 0.000, B 0.000, C 0.000 }
gfCNCPoint4[11674] = {X 140.7984, Y 77.7472, Z -5.5000, A 0.000, B 0.000, C 0.000 }
gfCNCPoint4[11675] = {X 155.8334, Y 61.2367, Z -5.5000, A 0.000, B 0.000, C 0.000 }
gfCNCPoint4[11676] = {X 155.4564, Y 60.5303, Z -5.5000, A 0.000, B 0.000, C 0.000 }
gfCNCPoint4[11677] = {X 155.2217, Y 59.7647, Z -5.5000, A 0.000, B 0.000, C 0.000 }
gfCNCPoint4[11678] = {X 155.1381, Y 58.9684, Z -5.5000, A 0.000, B 0.000, C 0.000 }
gfCNCPoint4[11679] = {X 155.1380, Y 58.0000, Z -5.5000, A 0.000, B 0.000, C 0.000 }
gfCNCPoint4[11680] = {X 155.2423, Y 57.0743, Z -5.5000, A 0.000, B 0.000, C 0.000 }
gfCNCPoint4[11681] = {X 155.5499, Y 56.1950, Z -5.5000, A 0.000, B 0.000, C 0.000 }
gfCNCPoint4[11682] = {X 156.0455, Y 55.4063, Z -5.5000, A 0.000, B 0.000, C 0.000 }
gfCNCPoint4[11683] = {X 156.7042, Y 54.7476, Z -5.5000, A 0.000, B 0.000, C 0.000 }
gfCNCPoint4[11684] = {X 157.4930, Y 54.2520, Z -5.5000, A 0.000, B 0.000, C 0.000 }
gfCNCPoint4[11685] = {X 158.3723, Y 53.9443, Z -5.5000, A 0.000, B 0.000, C 0.000 }
gfCNCPoint4[11686] = {X 159.2980, Y 53.8400, Z -5.5000, A 0.000, B 0.000, C 0.000 }
gfCNCPoint4[11687] = {X 178.5335, Y 53.8400, Z -5.5000, A 0.000, B 0.000, C 0.000 }
gfCNCPoint4[11688] = {X 179.4592, Y 53.9443, Z -5.5000, A 0.000, B 0.000, C 0.000 }
gfCNCPoint4[11689] = {X 180.3385, Y 54.2520, Z -5.5000, A 0.000, B 0.000, C 0.000 }
gfCNCPoint4[11690] = {X 181.1272, Y 54.7476, Z -5.5000, A 0.000, B 0.000, C 0.000 }
gfCNCPoint4[11691] = {X 181.7859, Y 55.4063, Z -5.5000, A 0.000, B 0.000, C 0.000 }
gfCNCPoint4[11692] = {X 182.2815, Y 56.1950, Z -5.5000, A 0.000, B 0.000, C 0.000 }
gfCNCPoint4[11693] = {X 182.5892, Y 57.0743, Z -5.5000, A 0.000, B 0.000, C 0.000 }
gfCNCPoint4[11694] = {X 182.6935, Y 58.0000, Z -5.5000, A 0.000, B 0.000, C 0.000 }
gfCNCPoint4[11695] = {X 182.6935, Y 58.9342, Z -5.5000, A 0.000, B 0.000, C 0.000 }
gfCNCPoint4[11696] = {X 182.6160, Y 59.7333, Z -5.5000, A 0.000, B 0.000, C 0.000 }
gfCNCPoint4[11697] = {X 182.3864, Y 60.5027, Z -5.5000, A 0.000, B 0.000, C 0.000 }
gfCNCPoint4[11698] = {X 182.0133, Y 61.2136, Z -5.5000, A 0.000, B 0.000, C 0.000 }
gfCNCPoint4[11699] = {X 209.3612, Y 91.0623, Z -5.5000, A 0.000, B 0.000, C 0.000 }
gfCNCPoint4[11700] = {X 210.0262, Y 91.7370, Z -5.5000, A 0.000, B 0.000, C 0.000 }
gfCNCPoint4[11701] = {X 210.7385, Y 92.3615, Z -5.5000, A 0.000, B 0.000, C 0.000 }
gfCNCPoint4[11702] = {X 211.0468, Y 92.5563, Z -5.5000, A 0.000, B 0.000, C 0.000 }
gfCNCPoint4[11703] = {X 211.3924, Y 92.6724, Z -5.5000, A 0.000, B 0.000, C 0.000 }
gfCNCPoint4[11704] = {X 213.3994, Y 92.9854, Z -5.5000, A 0.000, B 0.000, C 0.000 }
gfCNCPoint4[11705] = {X 214.4547, Y 92.8959, Z -5.5000, A 0.000, B 0.000, C 0.000 }
gfCNCPoint4[11706] = {X 215.5121, Y 92.8352, Z -5.5000, A 0.000, B 0.000, C 0.000 }
gfCNCPoint4[11707] = {X 216.2109, Y 92.7586, Z -5.5000, A 0.000, B 0.000, C 0.000 }
gfCNCPoint4[11708] = {X 216.8837, Y 92.5549, Z -5.5000, A 0.000, B 0.000, C 0.000 }
gfCNCPoint4[11709] = {X 217.5077, Y 92.2312, Z -5.5000, A 0.000, B 0.000, C 0.000 }
gfCNCPoint4[11710] = {X 223.0478, Y 88.6559, Z -5.5000, A 0.000, B 0.000, C 0.000 }
gfCNCPoint4[11711] = {X 246.1784, Y 73.8653, Z -5.5000, A 0.000, B 0.000, C 0.000 }
gfCNCPoint4[11712] = {X 221.6899, Y 64.2555, Z -5.5000, A 0.000, B 0.000, C 0.000 }
gfCNCPoint4[11713] = {X 219.9051, Y 63.6581, Z -5.5000, A 0.000, B 0.000, C 0.000 }
gfCNCPoint4[11714] = {X 218.0638, Y 63.2684, Z -5.5000, A 0.000, B 0.000, C 0.000 }
gfCNCPoint4[11715] = {X 216.1900, Y 63.0917, Z -5.5000, A 0.000, B 0.000, C 0.000 }
gfCNCPoint4[11716] = {X 215.2926, Y 62.9624, Z -5.5000, A 0.000, B 0.000, C 0.000 }
gfCNCPoint4[11717] = {X 214.4445, Y 62.6418, Z -5.5000, A 0.000, B 0.000, C 0.000 }
gfCNCPoint4[11718] = {X 213.6860, Y 62.1451, Z -5.5000, A 0.000, B 0.000, C 0.000 }
gfCNCPoint4[11719] = {X 213.0531, Y 61.4958, Z -5.5000, A 0.000, B 0.000, C 0.000 }
gfCNCPoint4[11720] = {X 212.5760, Y 60.7249, Z -5.5000, A 0.000, B 0.000, C 0.000 }
gfCNCPoint4[11721] = {X 212.2772, Y 59.8688, Z -5.5000, A 0.000, B 0.000, C 0.000 }
gfCNCPoint4[11722] = {X 212.1710, Y 58.9684, Z -5.5000, A 0.000, B 0.000, C 0.000 }
gfCNCPoint4[11723] = {X 212.1708, Y 58.0000, Z -5.5000, A 0.000, B 0.000, C 0.000 }
gfCNCPoint4[11724] = {X 212.2751, Y 57.0743, Z -5.5000, A 0.000, B 0.000, C 0.000 }
gfCNCPoint4[11725] = {X 212.5828, Y 56.1950, Z -5.5000, A 0.000, B 0.000, C 0.000 }
gfCNCPoint4[11726] = {X 213.0784, Y 55.4063, Z -5.5000, A 0.000, B 0.000, C 0.000 }
gfCNCPoint4[11727] = {X 213.7371, Y 54.7476, Z -5.5000, A 0.000, B 0.000, C 0.000 }
gfCNCPoint4[11728] = {X 214.5259, Y 54.2520, Z -5.5000, A 0.000, B 0.000, C 0.000 }
gfCNCPoint4[11729] = {X 215.4051, Y 53.9443, Z -5.5000, A 0.000, B 0.000, C 0.000 }
gfCNCPoint4[11730] = {X 216.3308, Y 53.8400, Z -5.5000, A 0.000, B 0.000, C 0.000 }
gfCNCPoint4[11731] = {X 237.2617, Y 53.8400, Z -5.5000, A 0.000, B 0.000, C 0.000 }
gfCNCPoint4[11732] = {X 238.1874, Y 53.9443, Z -5.5000, A 0.000, B 0.000, C 0.000 }
gfCNCPoint4[11733] = {X 239.0666, Y 54.2520, Z -5.5000, A 0.000, B 0.000, C 0.000 }
gfCNCPoint4[11734] = {X 239.8554, Y 54.7476, Z -5.5000, A 0.000, B 0.000, C 0.000 }
gfCNCPoint4[11735] = {X 240.5141, Y 55.4063, Z -5.5000, A 0.000, B 0.000, C 0.000 }
gfCNCPoint4[11736] = {X 241.0097, Y 56.1950, Z -5.5000, A 0.000, B 0.000, C 0.000 }
gfCNCPoint4[11737] = {X 241.3174, Y 57.0743, Z -5.5000, A 0.000, B 0.000, C 0.000 }
gfCNCPoint4[11738] = {X 241.4217, Y 58.0000, Z -5.5000, A 0.000, B 0.000, C 0.000 }
gfCNCPoint4[11739] = {X 241.4217, Y 58.3415, Z -5.5000, A 0.000, B 0.000, C 0.000 }
gfCNCPoint4[11740] = {X 248.0556, Y 60.9282, Z -5.5000, A 0.000, B 0.000, C 0.000 }
gfCNCPoint4[11741] = {X 275.7925, Y 71.9375, Z -5.5000, A 0.000, B 0.000, C 0.000 }
gfCNCPoint4[11742] = {X 275.7938, Y 63.0709, Z -5.5000, A 0.000, B 0.000, C 0.000 }
gfCNCPoint4[11743] = {X 275.6913, Y 63.0587, Z -5.5000, A 0.000, B 0.000, C 0.000 }
gfCNCPoint4[11744] = {X 275.5892, Y 63.0440, Z -5.5000, A 0.000, B 0.000, C 0.000 }
gfCNCPoint4[11745] = {X 274.6517, Y 62.7819, Z -5.5000, A 0.000, B 0.000, C 0.000 }
gfCNCPoint4[11746] = {X 273.8007, Y 62.3092, Z -5.5000, A 0.000, B 0.000, C 0.000 }
gfCNCPoint4[11747] = {X 273.0830, Y 61.6516, Z -5.5000, A 0.000, B 0.000, C 0.000 }
gfCNCPoint4[11748] = {X 272.5377, Y 60.8452, Z -5.5000, A 0.000, B 0.000, C 0.000 }
gfCNCPoint4[11749] = {X 272.1947, Y 59.9342, Z -5.5000, A 0.000, B 0.000, C 0.000 }
gfCNCPoint4[11750] = {X 272.0728, Y 58.9684, Z -5.5000, A 0.000, B 0.000, C 0.000 }
gfCNCPoint4[11751] = {X 272.0727, Y 58.0000, Z -5.5000, A 0.000, B 0.000, C 0.000 }
gfCNCPoint4[11752] = {X 272.1770, Y 57.0743, Z -5.5000, A 0.000, B 0.000, C 0.000 }
gfCNCPoint4[11753] = {X 272.4847, Y 56.1950, Z -5.5000, A 0.000, B 0.000, C 0.000 }
gfCNCPoint4[11754] = {X 272.9803, Y 55.4063, Z -5.5000, A 0.000, B 0.000, C 0.000 }
gfCNCPoint4[11755] = {X 273.6390, Y 54.7476, Z -5.5000, A 0.000, B 0.000, C 0.000 }
gfCNCPoint4[11756] = {X 274.4277, Y 54.2520, Z -5.5000, A 0.000, B 0.000, C 0.000 }
gfCNCPoint4[11757] = {X 275.3070, Y 53.9443, Z -5.5000, A 0.000, B 0.000, C 0.000 }
gfCNCPoint4[11758] = {X 276.2327, Y 53.8400, Z -5.5000, A 0.000, B 0.000, C 0.000 }
gfCNCPoint4[11759] = {X 292.7731, Y 53.8400, Z -5.5000, A 0.000, B 0.000, C 0.000 }
gfCNCPoint4[11760] = {X 293.6988, Y 53.9443, Z -5.5000, A 0.000, B 0.000, C 0.000 }
gfCNCPoint4[11761] = {X 294.5780, Y 54.2520, Z -5.5000, A 0.000, B 0.000, C 0.000 }
gfCNCPoint4[11762] = {X 295.3668, Y 54.7476, Z -5.5000, A 0.000, B 0.000, C 0.000 }
gfCNCPoint4[11763] = {X 296.0255, Y 55.4063, Z -5.5000, A 0.000, B 0.000, C 0.000 }
gfCNCPoint4[11764] = {X 296.5211, Y 56.1950, Z -5.5000, A 0.000, B 0.000, C 0.000 }
gfCNCPoint4[11765] = {X 296.8288, Y 57.0743, Z -5.5000, A 0.000, B 0.000, C 0.000 }
gfCNCPoint4[11766] = {X 296.9331, Y 58.0000, Z -5.5000, A 0.000, B 0.000, C 0.000 }
gfCNCPoint4[11767] = {X 296.9331, Y 58.9346, Z -5.5000, A 0.000, B 0.000, C 0.000 }
gfCNCPoint4[11768] = {X 296.8155, Y 59.9063, Z -5.5000, A 0.000, B 0.000, C 0.000 }
gfCNCPoint4[11769] = {X 296.4749, Y 60.8240, Z -5.5000, A 0.000, B 0.000, C 0.000 }
gfCNCPoint4[11770] = {X 295.9301, Y 61.6371, Z -5.5000, A 0.000, B 0.000, C 0.000 }
gfCNCPoint4[11771] = {X 295.2110, Y 62.3012, Z -5.5000, A 0.000, B 0.000, C 0.000 }
gfCNCPoint4[11772] = {X 294.3571, Y 62.7796, Z -5.5000, A 0.000, B 0.000, C 0.000 }
gfCNCPoint4[11773] = {X 293.4153, Y 63.0462, Z -5.5000, A 0.000, B 0.000, C 0.000 }
gfCNCPoint4[11774] = {X 293.3186, Y 63.0604, Z -5.5000, A 0.000, B 0.000, C 0.000 }
gfCNCPoint4[11775] = {X 293.2217, Y 63.0725, Z -5.5000, A 0.000, B 0.000, C 0.000 }
gfCNCPoint4[11776] = {X 293.2131, Y 63.1617, Z -5.5000, A 0.000, B 0.000, C 0.000 }
gfCNCPoint4[11777] = {X 293.2247, Y 92.9209, Z -5.5000, A 0.000, B 0.000, C 0.000 }
gfCNCPoint4[11778] = {X 293.3197, Y 92.9331, Z -5.5000, A 0.000, B 0.000, C 0.000 }
gfCNCPoint4[11779] = {X 293.4145, Y 92.9474, Z -5.5000, A 0.000, B 0.000, C 0.000 }
gfCNCPoint4[11780] = {X 294.3560, Y 93.2166, Z -5.5000, A 0.000, B 0.000, C 0.000 }
gfCNCPoint4[11781] = {X 295.2093, Y 93.6968, Z -5.5000, A 0.000, B 0.000, C 0.000 }
gfCNCPoint4[11782] = {X 295.9280, Y 94.3619, Z -5.5000, A 0.000, B 0.000, C 0.000 }
gfCNCPoint4[11783] = {X 296.4728, Y 95.1755, Z -5.5000, A 0.000, B 0.000, C 0.000 }
gfCNCPoint4[11784] = {X 296.8140, Y 96.0933, Z -5.5000, A 0.000, B 0.000, C 0.000 }
gfCNCPoint4[11785] = {X 296.9331, Y 97.0653, Z -5.5000, A 0.000, B 0.000, C 0.000 }
gfCNCPoint4[11786] = {X 296.9331, Y 98.0000, Z -5.5000, A 0.000, B 0.000, C 0.000 }
gfCNCPoint4[11787] = {X 296.8288, Y 98.9257, Z -5.5000, A 0.000, B 0.000, C 0.000 }
gfCNCPoint4[11788] = {X 296.5211, Y 99.8050, Z -5.5000, A 0.000, B 0.000, C 0.000 }
gfCNCPoint4[11789] = {X 296.0255, Y 100.5937, Z -5.5000, A 0.000, B 0.000, C 0.000 }
gfCNCPoint4[11790] = {X 295.3668, Y 101.2524, Z -5.5000, A 0.000, B 0.000, C 0.000 }
gfCNCPoint4[11791] = {X 294.5780, Y 101.7480, Z -5.5000, A 0.000, B 0.000, C 0.000 }
gfCNCPoint4[11792] = {X 293.6988, Y 102.0557, Z -5.5000, A 0.000, B 0.000, C 0.000 }
gfCNCPoint4[11793] = {X 292.7731, Y 102.1600, Z -5.5000, A 0.000, B 0.000, C 0.000 }
gfCNCPoint4[11794] = {X 276.2327, Y 102.1600, Z -5.5000, A 0.000, B 0.000, C 0.000 }
gfCNCPoint4[11795] = {X 275.3070, Y 102.0557, Z -5.5000, A 0.000, B 0.000, C 0.000 }
gfCNCPoint4[11796] = {X 274.4277, Y 101.7480, Z -5.5000, A 0.000, B 0.000, C 0.000 }
gfCNCPoint4[11797] = {X 273.6390, Y 101.2524, Z -5.5000, A 0.000, B 0.000, C 0.000 }
gfCNCPoint4[11798] = {X 272.9803, Y 100.5937, Z -5.5000, A 0.000, B 0.000, C 0.000 }
gfCNCPoint4[11799] = {X 272.4847, Y 99.8050, Z -5.5000, A 0.000, B 0.000, C 0.000 }
gfCNCPoint4[11800] = {X 272.1770, Y 98.9257, Z -5.5000, A 0.000, B 0.000, C 0.000 }
gfCNCPoint4[11801] = {X 272.0727, Y 98.0000, Z -5.5000, A 0.000, B 0.000, C 0.000 }
gfCNCPoint4[11802] = {X 272.0727, Y 97.0659, Z -5.5000, A 0.000, B 0.000, C 0.000 }
gfCNCPoint4[11803] = {X 272.1634, Y 96.2022, Z -5.5000, A 0.000, B 0.000, C 0.000 }
gfCNCPoint4[11804] = {X 272.4314, Y 95.3761, Z -5.5000, A 0.000, B 0.000, C 0.000 }
gfCNCPoint4[11805] = {X 272.8651, Y 94.6237, Z -5.5000, A 0.000, B 0.000, C 0.000 }
gfCNCPoint4[11806] = {X 273.4455, Y 93.9777, Z -5.5000, A 0.000, B 0.000, C 0.000 }
gfCNCPoint4[11807] = {X 274.1474, Y 93.4663, Z -5.5000, A 0.000, B 0.000, C 0.000 }
gfCNCPoint4[11808] = {X 274.9403, Y 93.1118, Z -5.5000, A 0.000, B 0.000, C 0.000 }
gfCNCPoint4[11809] = {X 275.7894, Y 92.9296, Z -5.5000, A 0.000, B 0.000, C 0.000 }
gfCNCPoint4[11810] = {X 275.7894, Y 85.4858, Z -5.5000, A 0.000, B 0.000, C 0.000 }
gfCNCPoint4[11811] = {X 262.6228, Y 80.3245, Z -5.5000, A 0.000, B 0.000, C 0.000 }
gfCNCPoint4[11812] = {X 262.1912, Y 80.5968, Z -5.5000, A 0.000, B 0.000, C 0.000 }
gfCNCPoint4[11813] = {X 237.6364, Y 96.5016, Z -5.5000, A 0.000, B 0.000, C 0.000 }
gfCNCPoint4[11814] = {X 237.6398, Y 97.0654, Z -5.5000, A 0.000, B 0.000, C 0.000 }
gfCNCPoint4[11815] = {X 237.6398, Y 98.0000, Z -5.5000, A 0.000, B 0.000, C 0.000 }
gfCNCPoint4[11816] = {X 237.5355, Y 98.9257, Z -5.5000, A 0.000, B 0.000, C 0.000 }
gfCNCPoint4[11817] = {X 237.2278, Y 99.8050, Z -5.5000, A 0.000, B 0.000, C 0.000 }
gfCNCPoint4[11818] = {X 236.7322, Y 100.5937, Z -5.5000, A 0.000, B 0.000, C 0.000 }
gfCNCPoint4[11819] = {X 236.0735, Y 101.2524, Z -5.5000, A 0.000, B 0.000, C 0.000 }
gfCNCPoint4[11820] = {X 235.2847, Y 101.7480, Z -5.5000, A 0.000, B 0.000, C 0.000 }
gfCNCPoint4[11821] = {X 234.4055, Y 102.0557, Z -5.5000, A 0.000, B 0.000, C 0.000 }
gfCNCPoint4[11822] = {X 233.4798, Y 102.1600, Z -5.5000, A 0.000, B 0.000, C 0.000 }
gfCNCPoint4[11823] = {X 214.1790, Y 102.1600, Z -5.5000, A 0.000, B 0.000, C 0.000 }
gfCNCPoint4[11824] = {X 213.7860, Y 102.1414, Z -5.5000, A 0.000, B 0.000, C 0.000 }
gfCNCPoint4[11825] = {X 213.3966, Y 102.0857, Z -5.5000, A 0.000, B 0.000, C 0.000 }
gfCNCPoint4[11826] = {X 213.0071, Y 102.1414, Z -5.5000, A 0.000, B 0.000, C 0.000 }
gfCNCPoint4[11827] = {X 212.6141, Y 102.1600, Z -5.5000, A 0.000, B 0.000, C 0.000 }
gfCNCPoint4[11828] = {X 194.9870, Y 102.1600, Z -5.5000, A 0.000, B 0.000, C 0.000 }
gfCNCPoint4[11829] = {X 194.0613, Y 102.0557, Z -5.5000, A 0.000, B 0.000, C 0.000 }
gfCNCPoint4[11830] = {X 193.1820, Y 101.7480, Z -5.5000, A 0.000, B 0.000, C 0.000 }
gfCNCPoint4[11831] = {X 192.3932, Y 101.2524, Z -5.5000, A 0.000, B 0.000, C 0.000 }
gfCNCPoint4[11832] = {X 191.7345, Y 100.5937, Z -5.5000, A 0.000, B 0.000, C 0.000 }
gfCNCPoint4[11833] = {X 191.2389, Y 99.8050, Z -5.5000, A 0.000, B 0.000, C 0.000 }
gfCNCPoint4[11834] = {X 190.9313, Y 98.9257, Z -5.5000, A 0.000, B 0.000, C 0.000 }
gfCNCPoint4[11835] = {X 190.8270, Y 98.0000, Z -5.5000, A 0.000, B 0.000, C 0.000 }
gfCNCPoint4[11836] = {X 190.8270, Y 97.0659, Z -5.5000, A 0.000, B 0.000, C 0.000 }
gfCNCPoint4[11837] = {X 190.9241, Y 96.1723, Z -5.5000, A 0.000, B 0.000, C 0.000 }
gfCNCPoint4[11838] = {X 191.2109, Y 95.3203, Z -5.5000, A 0.000, B 0.000, C 0.000 }
gfCNCPoint4[11839] = {X 191.6741, Y 94.5499, Z -5.5000, A 0.000, B 0.000, C 0.000 }
gfCNCPoint4[11840] = {X 191.7354, Y 94.4712, Z -5.5000, A 0.000, B 0.000, C 0.000 }
gfCNCPoint4[11841] = {X 191.7986, Y 94.3939, Z -5.5000, A 0.000, B 0.000, C 0.000 }
gfCNCPoint4[11842] = {X 188.6351, Y 90.9402, Z -5.5000, A 0.000, B 0.000, C 0.000 }
gfCNCPoint4[11843] = {X 150.0187, Y 90.9402, Z -5.5000, A 0.000, B 0.000, C 0.000 }
gfCNCPoint4[11844] = {X 146.9337, Y 94.3580, Z -5.5000, A 0.000, B 0.000, C 0.000 }
gfCNCPoint4[11845] = {X 147.4796, Y 95.1727, Z -5.5000, A 0.000, B 0.000, C 0.000 }
gfCNCPoint4[11846] = {X 147.8210, Y 96.0920, Z -5.5000, A 0.000, B 0.000, C 0.000 }
gfCNCPoint4[11847] = {X 147.9391, Y 97.0655, Z -5.5000, A 0.000, B 0.000, C 0.000 }
gfCNCPoint4[11848] = {X 147.9391, Y 98.0000, Z -5.5000, A 0.000, B 0.000, C 0.000 }
gfCNCPoint4[11849] = {X 147.8348, Y 98.9257, Z -5.5000, A 0.000, B 0.000, C 0.000 }
gfCNCPoint4[11850] = {X 147.5271, Y 99.8050, Z -5.5000, A 0.000, B 0.000, C 0.000 }
gfCNCPoint4[11851] = {X 147.0315, Y 100.5937, Z -5.5000, A 0.000, B 0.000, C 0.000 }
gfCNCPoint4[11852] = {X 146.3728, Y 101.2524, Z -5.5000, A 0.000, B 0.000, C 0.000 }
gfCNCPoint4[11853] = {X 145.5841, Y 101.7480, Z -5.5000, A 0.000, B 0.000, C 0.000 }
gfCNCPoint4[11854] = {X 144.7048, Y 102.0557, Z -5.5000, A 0.000, B 0.000, C 0.000 }
gfCNCPoint4[11855] = {X 143.7791, Y 102.1600, Z -5.5000, A 0.000, B 0.000, C 0.000 }
gfCNCPoint4[11856] = {X 125.0000, Y 102.1600, Z -5.5000, A 0.000, B 0.000, C 0.000 }
gfCNCPoint4[11857] = {X 124.0743, Y 102.0557, Z -5.5000, A 0.000, B 0.000, C 0.000 }
gfCNCPoint4[11858] = {X 123.1950, Y 101.7480, Z -5.5000, A 0.000, B 0.000, C 0.000 }
gfCNCPoint4[11859] = {X 122.4063, Y 101.2524, Z -5.5000, A 0.000, B 0.000, C 0.000 }
gfCNCPoint4[11860] = {X 121.7476, Y 100.5937, Z -5.5000, A 0.000, B 0.000, C 0.000 }
gfCNCPoint4[11861] = {X 121.2520, Y 99.8050, Z -5.5000, A 0.000, B 0.000, C 0.000 }
gfCNCPoint4[11862] = {X 120.9443, Y 98.9257, Z -5.5000, A 0.000, B 0.000, C 0.000 }
gfCNCPoint4[11863] = {X 120.8400, Y 98.0000, Z -5.5000, A 0.000, B 0.000, C 0.000 }
gfCNCPoint4[11864] = {X 120.8400, Y 97.0659, Z -5.5000, A 0.000, B 0.000, C 0.000 }
gfCNCPoint4[11865] = {X 120.9406, Y 96.1568, Z -5.5000, A 0.000, B 0.000, C 0.000 }
gfCNCPoint4[11866] = {X 121.2374, Y 95.2916, Z -5.5000, A 0.000, B 0.000, C 0.000 }
gfCNCPoint4[11867] = {X 121.7161, Y 94.5121, Z -5.5000, A 0.000, B 0.000, C 0.000 }
gfCNCPoint4[11868] = {X 122.3537, Y 93.8562, Z -5.5000, A 0.000, B 0.000, C 0.000 }
gfCNCPoint4[11869] = {X 123.1191, Y 93.3554, Z -5.5000, A 0.000, B 0.000, C 0.000 }
gfCNCPoint4[11870] = {X 123.9755, Y 93.0341, Z -5.5000, A 0.000, B 0.000, C 0.000 }
gfCNCPoint4[11871] = {X 124.8814, Y 92.9076, Z -5.5000, A 0.000, B 0.000, C 0.000 }
gfCNCPoint4[11872] = {X 124.9147, Y 92.8893, Z -5.5000, A 0.000, B 0.000, C 0.000 }
gfCNCPoint4[11873] = {X 124.9513, Y 92.8794, Z -5.5000, A 0.000, B 0.000, C 0.000 }
gfCNCPoint4[11874] = {X 125.4717, Y 92.8022, Z -5.5000, A 0.000, B 0.000, C 0.000 }
gfCNCPoint4[11875] = {X 126.3313, Y 92.6569, Z -5.5000, A 0.000, B 0.000, C 0.000 }
gfCNCPoint4[11876] = {X 127.1787, Y 92.4517, Z -5.5000, A 0.000, B 0.000, C 0.000 }
gfCNCPoint4[11877] = {X 128.4212, Y 91.2828, Z -5.5000, A 0.000, B 0.000, C 0.000 }
gfCNCPoint4[11878] = {X 129.5974, Y 90.0473, Z -5.5000, A 0.000, B 0.000, C 0.000 }
gfCNCPoint4[11879] = {X 140.7984, Y 77.7472, Z -5.5000, A 0.000, B 0.000, C 0.000 }
gfCNCPoint4[11880] = {X 137.8409, Y 75.0540, Z -5.5000, A 0.000, B 0.000, C 0.000 }
gfCNCPoint4[11881] = {X 140.8575, Y 77.8010, Z -5.5000, A 0.000, B 0.000, C 0.000 }
gfCNCPoint4[11882] = {X 155.9349, Y 61.2441, Z -5.5000, A 0.000, B 0.000, C 0.000 }
gfCNCPoint4[11883] = {X 155.5464, Y 60.5379, Z -5.5000, A 0.000, B 0.000, C 0.000 }
gfCNCPoint4[11884] = {X 155.3043, Y 59.7691, Z -5.5000, A 0.000, B 0.000, C 0.000 }
gfCNCPoint4[11885] = {X 155.2181, Y 58.9678, Z -5.5000, A 0.000, B 0.000, C 0.000 }
gfCNCPoint4[11886] = {X 155.2180, Y 58.0000, Z -5.5000, A 0.000, B 0.000, C 0.000 }
gfCNCPoint4[11887] = {X 155.3203, Y 57.0921, Z -5.5000, A 0.000, B 0.000, C 0.000 }
gfCNCPoint4[11888] = {X 155.6220, Y 56.2298, Z -5.5000, A 0.000, B 0.000, C 0.000 }
gfCNCPoint4[11889] = {X 156.1081, Y 55.4562, Z -5.5000, A 0.000, B 0.000, C 0.000 }
gfCNCPoint4[11890] = {X 156.7541, Y 54.8101, Z -5.5000, A 0.000, B 0.000, C 0.000 }
gfCNCPoint4[11891] = {X 157.5277, Y 54.3240, Z -5.5000, A 0.000, B 0.000, C 0.000 }
gfCNCPoint4[11892] = {X 158.3901, Y 54.0223, Z -5.5000, A 0.000, B 0.000, C 0.000 }
gfCNCPoint4[11893] = {X 159.2980, Y 53.9200, Z -5.5000, A 0.000, B 0.000, C 0.000 }
gfCNCPoint4[11894] = {X 178.5335, Y 53.9200, Z -5.5000, A 0.000, B 0.000, C 0.000 }
gfCNCPoint4[11895] = {X 179.4414, Y 54.0223, Z -5.5000, A 0.000, B 0.000, C 0.000 }
gfCNCPoint4[11896] = {X 180.3037, Y 54.3240, Z -5.5000, A 0.000, B 0.000, C 0.000 }
gfCNCPoint4[11897] = {X 181.0773, Y 54.8101, Z -5.5000, A 0.000, B 0.000, C 0.000 }
gfCNCPoint4[11898] = {X 181.7234, Y 55.4562, Z -5.5000, A 0.000, B 0.000, C 0.000 }
gfCNCPoint4[11899] = {X 182.2095, Y 56.2298, Z -5.5000, A 0.000, B 0.000, C 0.000 }
gfCNCPoint4[11900] = {X 182.5112, Y 57.0921, Z -5.5000, A 0.000, B 0.000, C 0.000 }
gfCNCPoint4[11901] = {X 182.6135, Y 58.0000, Z -5.5000, A 0.000, B 0.000, C 0.000 }
gfCNCPoint4[11902] = {X 182.6135, Y 58.9342, Z -5.5000, A 0.000, B 0.000, C 0.000 }
gfCNCPoint4[11903] = {X 182.5335, Y 59.7383, Z -5.5000, A 0.000, B 0.000, C 0.000 }
gfCNCPoint4[11904] = {X 182.2965, Y 60.5108, Z -5.5000, A 0.000, B 0.000, C 0.000 }
gfCNCPoint4[11905] = {X 181.9120, Y 61.2214, Z -5.5000, A 0.000, B 0.000, C 0.000 }
gfCNCPoint4[11906] = {X 209.3023, Y 91.1164, Z -5.5000, A 0.000, B 0.000, C 0.000 }
gfCNCPoint4[11907] = {X 209.9713, Y 91.7952, Z -5.5000, A 0.000, B 0.000, C 0.000 }
gfCNCPoint4[11908] = {X 210.6880, Y 92.4235, Z -5.5000, A 0.000, B 0.000, C 0.000 }
gfCNCPoint4[11909] = {X 211.0133, Y 92.6290, Z -5.5000, A 0.000, B 0.000, C 0.000 }
gfCNCPoint4[11910] = {X 211.3782, Y 92.7511, Z -5.5000, A 0.000, B 0.000, C 0.000 }
gfCNCPoint4[11911] = {X 213.3972, Y 93.0660, Z -5.5000, A 0.000, B 0.000, C 0.000 }
gfCNCPoint4[11912] = {X 214.4548, Y 92.9761, Z -5.5000, A 0.000, B 0.000, C 0.000 }
gfCNCPoint4[11913] = {X 215.5145, Y 92.9151, Z -5.5000, A 0.000, B 0.000, C 0.000 }
gfCNCPoint4[11914] = {X 216.2276, Y 92.8368, Z -5.5000, A 0.000, B 0.000, C 0.000 }
gfCNCPoint4[11915] = {X 216.9142, Y 92.6289, Z -5.5000, A 0.000, B 0.000, C 0.000 }
gfCNCPoint4[11916] = {X 217.5510, Y 92.2985, Z -5.5000, A 0.000, B 0.000, C 0.000 }
gfCNCPoint4[11917] = {X 223.0910, Y 88.7232, Z -5.5000, A 0.000, B 0.000, C 0.000 }
gfCNCPoint4[11918] = {X 246.3537, Y 73.8482, Z -5.5000, A 0.000, B 0.000, C 0.000 }
gfCNCPoint4[11919] = {X 221.7196, Y 64.1812, Z -5.5000, A 0.000, B 0.000, C 0.000 }
gfCNCPoint4[11920] = {X 219.9261, Y 63.5809, Z -5.5000, A 0.000, B 0.000, C 0.000 }
gfCNCPoint4[11921] = {X 218.0758, Y 63.1894, Z -5.5000, A 0.000, B 0.000, C 0.000 }
gfCNCPoint4[11922] = {X 216.1929, Y 63.0117, Z -5.5000, A 0.000, B 0.000, C 0.000 }
gfCNCPoint4[11923] = {X 215.3127, Y 62.8850, Z -5.5000, A 0.000, B 0.000, C 0.000 }
gfCNCPoint4[11924] = {X 214.4809, Y 62.5706, Z -5.5000, A 0.000, B 0.000, C 0.000 }
gfCNCPoint4[11925] = {X 213.7369, Y 62.0834, Z -5.5000, A 0.000, B 0.000, C 0.000 }
gfCNCPoint4[11926] = {X 213.1162, Y 61.4466, Z -5.5000, A 0.000, B 0.000, C 0.000 }
gfCNCPoint4[11927] = {X 212.6482, Y 60.6905, Z -5.5000, A 0.000, B 0.000, C 0.000 }
gfCNCPoint4[11928] = {X 212.3552, Y 59.8509, Z -5.5000, A 0.000, B 0.000, C 0.000 }
gfCNCPoint4[11929] = {X 212.2509, Y 58.9678, Z -5.5000, A 0.000, B 0.000, C 0.000 }
gfCNCPoint4[11930] = {X 212.2508, Y 58.0000, Z -5.5000, A 0.000, B 0.000, C 0.000 }
gfCNCPoint4[11931] = {X 212.3531, Y 57.0921, Z -5.5000, A 0.000, B 0.000, C 0.000 }
gfCNCPoint4[11932] = {X 212.6549, Y 56.2298, Z -5.5000, A 0.000, B 0.000, C 0.000 }
gfCNCPoint4[11933] = {X 213.1409, Y 55.4562, Z -5.5000, A 0.000, B 0.000, C 0.000 }
gfCNCPoint4[11934] = {X 213.7870, Y 54.8101, Z -5.5000, A 0.000, B 0.000, C 0.000 }
gfCNCPoint4[11935] = {X 214.5606, Y 54.3240, Z -5.5000, A 0.000, B 0.000, C 0.000 }
gfCNCPoint4[11936] = {X 215.4229, Y 54.0223, Z -5.5000, A 0.000, B 0.000, C 0.000 }
gfCNCPoint4[11937] = {X 216.3308, Y 53.9200, Z -5.5000, A 0.000, B 0.000, C 0.000 }
gfCNCPoint4[11938] = {X 237.2617, Y 53.9200, Z -5.5000, A 0.000, B 0.000, C 0.000 }
gfCNCPoint4[11939] = {X 238.1696, Y 54.0223, Z -5.5000, A 0.000, B 0.000, C 0.000 }
gfCNCPoint4[11940] = {X 239.0319, Y 54.3240, Z -5.5000, A 0.000, B 0.000, C 0.000 }
gfCNCPoint4[11941] = {X 239.8055, Y 54.8101, Z -5.5000, A 0.000, B 0.000, C 0.000 }
gfCNCPoint4[11942] = {X 240.4516, Y 55.4562, Z -5.5000, A 0.000, B 0.000, C 0.000 }
gfCNCPoint4[11943] = {X 240.9376, Y 56.2298, Z -5.5000, A 0.000, B 0.000, C 0.000 }
gfCNCPoint4[11944] = {X 241.2394, Y 57.0921, Z -5.5000, A 0.000, B 0.000, C 0.000 }
gfCNCPoint4[11945] = {X 241.3417, Y 58.0000, Z -5.5000, A 0.000, B 0.000, C 0.000 }
gfCNCPoint4[11946] = {X 241.3417, Y 58.3961, Z -5.5000, A 0.000, B 0.000, C 0.000 }
gfCNCPoint4[11947] = {X 248.0263, Y 61.0026, Z -5.5000, A 0.000, B 0.000, C 0.000 }
gfCNCPoint4[11948] = {X 275.8725, Y 72.0553, Z -5.5000, A 0.000, B 0.000, C 0.000 }
gfCNCPoint4[11949] = {X 275.8738, Y 62.9983, Z -5.5000, A 0.000, B 0.000, C 0.000 }
gfCNCPoint4[11950] = {X 275.7374, Y 62.9839, Z -5.5000, A 0.000, B 0.000, C 0.000 }
gfCNCPoint4[11951] = {X 275.6015, Y 62.9650, Z -5.5000, A 0.000, B 0.000, C 0.000 }
gfCNCPoint4[11952] = {X 274.6821, Y 62.7079, Z -5.5000, A 0.000, B 0.000, C 0.000 }
gfCNCPoint4[11953] = {X 273.8475, Y 62.2443, Z -5.5000, A 0.000, B 0.000, C 0.000 }
gfCNCPoint4[11954] = {X 273.1436, Y 61.5993, Z -5.5000, A 0.000, B 0.000, C 0.000 }
gfCNCPoint4[11955] = {X 272.6087, Y 60.8085, Z -5.5000, A 0.000, B 0.000, C 0.000 }
gfCNCPoint4[11956] = {X 272.2724, Y 59.9150, Z -5.5000, A 0.000, B 0.000, C 0.000 }
gfCNCPoint4[11957] = {X 272.1528, Y 58.9678, Z -5.5000, A 0.000, B 0.000, C 0.000 }
gfCNCPoint4[11958] = {X 272.1527, Y 58.0000, Z -5.5000, A 0.000, B 0.000, C 0.000 }
gfCNCPoint4[11959] = {X 272.2550, Y 57.0921, Z -5.5000, A 0.000, B 0.000, C 0.000 }
gfCNCPoint4[11960] = {X 272.5567, Y 56.2298, Z -5.5000, A 0.000, B 0.000, C 0.000 }
gfCNCPoint4[11961] = {X 273.0428, Y 55.4562, Z -5.5000, A 0.000, B 0.000, C 0.000 }
gfCNCPoint4[11962] = {X 273.6889, Y 54.8101, Z -5.5000, A 0.000, B 0.000, C 0.000 }
gfCNCPoint4[11963] = {X 274.4624, Y 54.3240, Z -5.5000, A 0.000, B 0.000, C 0.000 }
gfCNCPoint4[11964] = {X 275.3248, Y 54.0223, Z -5.5000, A 0.000, B 0.000, C 0.000 }
gfCNCPoint4[11965] = {X 276.2327, Y 53.9200, Z -5.5000, A 0.000, B 0.000, C 0.000 }
gfCNCPoint4[11966] = {X 292.7731, Y 53.9200, Z -5.5000, A 0.000, B 0.000, C 0.000 }
gfCNCPoint4[11967] = {X 293.6810, Y 54.0223, Z -5.5000, A 0.000, B 0.000, C 0.000 }
gfCNCPoint4[11968] = {X 294.5433, Y 54.3240, Z -5.5000, A 0.000, B 0.000, C 0.000 }
gfCNCPoint4[11969] = {X 295.3169, Y 54.8101, Z -5.5000, A 0.000, B 0.000, C 0.000 }
gfCNCPoint4[11970] = {X 295.9630, Y 55.4562, Z -5.5000, A 0.000, B 0.000, C 0.000 }
gfCNCPoint4[11971] = {X 296.4490, Y 56.2298, Z -5.5000, A 0.000, B 0.000, C 0.000 }
gfCNCPoint4[11972] = {X 296.7508, Y 57.0921, Z -5.5000, A 0.000, B 0.000, C 0.000 }
gfCNCPoint4[11973] = {X 296.8531, Y 58.0000, Z -5.5000, A 0.000, B 0.000, C 0.000 }
gfCNCPoint4[11974] = {X 296.8531, Y 58.9343, Z -5.5000, A 0.000, B 0.000, C 0.000 }
gfCNCPoint4[11975] = {X 296.7377, Y 59.8874, Z -5.5000, A 0.000, B 0.000, C 0.000 }
gfCNCPoint4[11976] = {X 296.4037, Y 60.7875, Z -5.5000, A 0.000, B 0.000, C 0.000 }
gfCNCPoint4[11977] = {X 295.8693, Y 61.5851, Z -5.5000, A 0.000, B 0.000, C 0.000 }
gfCNCPoint4[11978] = {X 295.1640, Y 62.2365, Z -5.5000, A 0.000, B 0.000, C 0.000 }
gfCNCPoint4[11979] = {X 294.3264, Y 62.7057, Z -5.5000, A 0.000, B 0.000, C 0.000 }
gfCNCPoint4[11980] = {X 293.4026, Y 62.9672, Z -5.5000, A 0.000, B 0.000, C 0.000 }
gfCNCPoint4[11981] = {X 293.2758, Y 62.9854, Z -5.5000, A 0.000, B 0.000, C 0.000 }
gfCNCPoint4[11982] = {X 293.1484, Y 62.9997, Z -5.5000, A 0.000, B 0.000, C 0.000 }
gfCNCPoint4[11983] = {X 293.1331, Y 63.1579, Z -5.5000, A 0.000, B 0.000, C 0.000 }
gfCNCPoint4[11984] = {X 293.1447, Y 92.9928, Z -5.5000, A 0.000, B 0.000, C 0.000 }
gfCNCPoint4[11985] = {X 293.2734, Y 93.0076, Z -5.5000, A 0.000, B 0.000, C 0.000 }
gfCNCPoint4[11986] = {X 293.4017, Y 93.0264, Z -5.5000, A 0.000, B 0.000, C 0.000 }
gfCNCPoint4[11987] = {X 294.3252, Y 93.2904, Z -5.5000, A 0.000, B 0.000, C 0.000 }
gfCNCPoint4[11988] = {X 295.1622, Y 93.7615, Z -5.5000, A 0.000, B 0.000, C 0.000 }
gfCNCPoint4[11989] = {X 295.8672, Y 94.4139, Z -5.5000, A 0.000, B 0.000, C 0.000 }
gfCNCPoint4[11990] = {X 296.4016, Y 95.2120, Z -5.5000, A 0.000, B 0.000, C 0.000 }
gfCNCPoint4[11991] = {X 296.7363, Y 96.1123, Z -5.5000, A 0.000, B 0.000, C 0.000 }
gfCNCPoint4[11992] = {X 296.8531, Y 97.0657, Z -5.5000, A 0.000, B 0.000, C 0.000 }
gfCNCPoint4[11993] = {X 296.8531, Y 98.0000, Z -5.5000, A 0.000, B 0.000, C 0.000 }
gfCNCPoint4[11994] = {X 296.7508, Y 98.9079, Z -5.5000, A 0.000, B 0.000, C 0.000 }
gfCNCPoint4[11995] = {X 296.4490, Y 99.7702, Z -5.5000, A 0.000, B 0.000, C 0.000 }
gfCNCPoint4[11996] = {X 295.9630, Y 100.5438, Z -5.5000, A 0.000, B 0.000, C 0.000 }
gfCNCPoint4[11997] = {X 295.3169, Y 101.1899, Z -5.5000, A 0.000, B 0.000, C 0.000 }
gfCNCPoint4[11998] = {X 294.5433, Y 101.6760, Z -5.5000, A 0.000, B 0.000, C 0.000 }
gfCNCPoint4[11999] = {X 293.6810, Y 101.9777, Z -5.5000, A 0.000, B 0.000, C 0.000 }
gfCNCPoint4[12000] = {X 292.7731, Y 102.0800, Z -5.5000, A 0.000, B 0.000, C 0.000 }
gfCNCPoint4[12001] = {X 276.2327, Y 102.0800, Z -5.5000, A 0.000, B 0.000, C 0.000 }
gfCNCPoint4[12002] = {X 275.3248, Y 101.9777, Z -5.5000, A 0.000, B 0.000, C 0.000 }
gfCNCPoint4[12003] = {X 274.4624, Y 101.6760, Z -5.5000, A 0.000, B 0.000, C 0.000 }
gfCNCPoint4[12004] = {X 273.6889, Y 101.1899, Z -5.5000, A 0.000, B 0.000, C 0.000 }
gfCNCPoint4[12005] = {X 273.0428, Y 100.5438, Z -5.5000, A 0.000, B 0.000, C 0.000 }
gfCNCPoint4[12006] = {X 272.5567, Y 99.7702, Z -5.5000, A 0.000, B 0.000, C 0.000 }
gfCNCPoint4[12007] = {X 272.2550, Y 98.9079, Z -5.5000, A 0.000, B 0.000, C 0.000 }
gfCNCPoint4[12008] = {X 272.1527, Y 98.0000, Z -5.5000, A 0.000, B 0.000, C 0.000 }
gfCNCPoint4[12009] = {X 272.1527, Y 97.0659, Z -5.5000, A 0.000, B 0.000, C 0.000 }
gfCNCPoint4[12010] = {X 272.2438, Y 96.2087, Z -5.5000, A 0.000, B 0.000, C 0.000 }
gfCNCPoint4[12011] = {X 272.5129, Y 95.3899, Z -5.5000, A 0.000, B 0.000, C 0.000 }
gfCNCPoint4[12012] = {X 272.9480, Y 94.6458, Z -5.5000, A 0.000, B 0.000, C 0.000 }
gfCNCPoint4[12013] = {X 273.5297, Y 94.0097, Z -5.5000, A 0.000, B 0.000, C 0.000 }
gfCNCPoint4[12014] = {X 274.2321, Y 93.5101, Z -5.5000, A 0.000, B 0.000, C 0.000 }
gfCNCPoint4[12015] = {X 275.0238, Y 93.1692, Z -5.5000, A 0.000, B 0.000, C 0.000 }
gfCNCPoint4[12016] = {X 275.8694, Y 93.0021, Z -5.5000, A 0.000, B 0.000, C 0.000 }
gfCNCPoint4[12017] = {X 275.8694, Y 85.4313, Z -5.5000, A 0.000, B 0.000, C 0.000 }
gfCNCPoint4[12018] = {X 262.6143, Y 80.2353, Z -5.5000, A 0.000, B 0.000, C 0.000 }
gfCNCPoint4[12019] = {X 262.1481, Y 80.5294, Z -5.5000, A 0.000, B 0.000, C 0.000 }
gfCNCPoint4[12020] = {X 237.5561, Y 96.4582, Z -5.5000, A 0.000, B 0.000, C 0.000 }
gfCNCPoint4[12021] = {X 237.5598, Y 97.0657, Z -5.5000, A 0.000, B 0.000, C 0.000 }
gfCNCPoint4[12022] = {X 237.5598, Y 98.0000, Z -5.5000, A 0.000, B 0.000, C 0.000 }
gfCNCPoint4[12023] = {X 237.4575, Y 98.9079, Z -5.5000, A 0.000, B 0.000, C 0.000 }
gfCNCPoint4[12024] = {X 237.1557, Y 99.7702, Z -5.5000, A 0.000, B 0.000, C 0.000 }
gfCNCPoint4[12025] = {X 236.6697, Y 100.5438, Z -5.5000, A 0.000, B 0.000, C 0.000 }
gfCNCPoint4[12026] = {X 236.0236, Y 101.1899, Z -5.5000, A 0.000, B 0.000, C 0.000 }
gfCNCPoint4[12027] = {X 235.2500, Y 101.6760, Z -5.5000, A 0.000, B 0.000, C 0.000 }
gfCNCPoint4[12028] = {X 234.3877, Y 101.9777, Z -5.5000, A 0.000, B 0.000, C 0.000 }
gfCNCPoint4[12029] = {X 233.4798, Y 102.0800, Z -5.5000, A 0.000, B 0.000, C 0.000 }
gfCNCPoint4[12030] = {X 214.1790, Y 102.0800, Z -5.5000, A 0.000, B 0.000, C 0.000 }
gfCNCPoint4[12031] = {X 213.7860, Y 102.0610, Z -5.5000, A 0.000, B 0.000, C 0.000 }
gfCNCPoint4[12032] = {X 213.3966, Y 102.0043, Z -5.5000, A 0.000, B 0.000, C 0.000 }
gfCNCPoint4[12033] = {X 213.0072, Y 102.0610, Z -5.5000, A 0.000, B 0.000, C 0.000 }
gfCNCPoint4[12034] = {X 212.6141, Y 102.0800, Z -5.5000, A 0.000, B 0.000, C 0.000 }
gfCNCPoint4[12035] = {X 194.9870, Y 102.0800, Z -5.5000, A 0.000, B 0.000, C 0.000 }
gfCNCPoint4[12036] = {X 194.0791, Y 101.9777, Z -5.5000, A 0.000, B 0.000, C 0.000 }
gfCNCPoint4[12037] = {X 193.2167, Y 101.6760, Z -5.5000, A 0.000, B 0.000, C 0.000 }
gfCNCPoint4[12038] = {X 192.4431, Y 101.1899, Z -5.5000, A 0.000, B 0.000, C 0.000 }
gfCNCPoint4[12039] = {X 191.7971, Y 100.5438, Z -5.5000, A 0.000, B 0.000, C 0.000 }
gfCNCPoint4[12040] = {X 191.3110, Y 99.7702, Z -5.5000, A 0.000, B 0.000, C 0.000 }
gfCNCPoint4[12041] = {X 191.0093, Y 98.9079, Z -5.5000, A 0.000, B 0.000, C 0.000 }
gfCNCPoint4[12042] = {X 190.9070, Y 98.0000, Z -5.5000, A 0.000, B 0.000, C 0.000 }
gfCNCPoint4[12043] = {X 190.9070, Y 97.0659, Z -5.5000, A 0.000, B 0.000, C 0.000 }
gfCNCPoint4[12044] = {X 191.0022, Y 96.1894, Z -5.5000, A 0.000, B 0.000, C 0.000 }
gfCNCPoint4[12045] = {X 191.2835, Y 95.3539, Z -5.5000, A 0.000, B 0.000, C 0.000 }
gfCNCPoint4[12046] = {X 191.7378, Y 94.5983, Z -5.5000, A 0.000, B 0.000, C 0.000 }
gfCNCPoint4[12047] = {X 191.8199, Y 94.4938, Z -5.5000, A 0.000, B 0.000, C 0.000 }
gfCNCPoint4[12048] = {X 191.9053, Y 94.3920, Z -5.5000, A 0.000, B 0.000, C 0.000 }
gfCNCPoint4[12049] = {X 188.6703, Y 90.8602, Z -5.5000, A 0.000, B 0.000, C 0.000 }
gfCNCPoint4[12050] = {X 149.9831, Y 90.8602, Z -5.5000, A 0.000, B 0.000, C 0.000 }
gfCNCPoint4[12051] = {X 146.8268, Y 94.3571, Z -5.5000, A 0.000, B 0.000, C 0.000 }
gfCNCPoint4[12052] = {X 147.3869, Y 95.1676, Z -5.5000, A 0.000, B 0.000, C 0.000 }
gfCNCPoint4[12053] = {X 147.7377, Y 96.0881, Z -5.5000, A 0.000, B 0.000, C 0.000 }
gfCNCPoint4[12054] = {X 147.8591, Y 97.0658, Z -5.5000, A 0.000, B 0.000, C 0.000 }
gfCNCPoint4[12055] = {X 147.8591, Y 98.0000, Z -5.5000, A 0.000, B 0.000, C 0.000 }
gfCNCPoint4[12056] = {X 147.7568, Y 98.9079, Z -5.5000, A 0.000, B 0.000, C 0.000 }
gfCNCPoint4[12057] = {X 147.4551, Y 99.7702, Z -5.5000, A 0.000, B 0.000, C 0.000 }
gfCNCPoint4[12058] = {X 146.9690, Y 100.5438, Z -5.5000, A 0.000, B 0.000, C 0.000 }
gfCNCPoint4[12059] = {X 146.3229, Y 101.1899, Z -5.5000, A 0.000, B 0.000, C 0.000 }
gfCNCPoint4[12060] = {X 145.5494, Y 101.6760, Z -5.5000, A 0.000, B 0.000, C 0.000 }
gfCNCPoint4[12061] = {X 144.6870, Y 101.9777, Z -5.5000, A 0.000, B 0.000, C 0.000 }
gfCNCPoint4[12062] = {X 143.7791, Y 102.0800, Z -5.5000, A 0.000, B 0.000, C 0.000 }
gfCNCPoint4[12063] = {X 125.0000, Y 102.0800, Z -5.5000, A 0.000, B 0.000, C 0.000 }
gfCNCPoint4[12064] = {X 124.0921, Y 101.9777, Z -5.5000, A 0.000, B 0.000, C 0.000 }
gfCNCPoint4[12065] = {X 123.2298, Y 101.6760, Z -5.5000, A 0.000, B 0.000, C 0.000 }
gfCNCPoint4[12066] = {X 122.4562, Y 101.1899, Z -5.5000, A 0.000, B 0.000, C 0.000 }
gfCNCPoint4[12067] = {X 121.8101, Y 100.5438, Z -5.5000, A 0.000, B 0.000, C 0.000 }
gfCNCPoint4[12068] = {X 121.3240, Y 99.7702, Z -5.5000, A 0.000, B 0.000, C 0.000 }
gfCNCPoint4[12069] = {X 121.0223, Y 98.9079, Z -5.5000, A 0.000, B 0.000, C 0.000 }
gfCNCPoint4[12070] = {X 120.9200, Y 98.0000, Z -5.5000, A 0.000, B 0.000, C 0.000 }
gfCNCPoint4[12071] = {X 120.9200, Y 97.0659, Z -5.5000, A 0.000, B 0.000, C 0.000 }
gfCNCPoint4[12072] = {X 121.0194, Y 96.1710, Z -5.5000, A 0.000, B 0.000, C 0.000 }
gfCNCPoint4[12073] = {X 121.3126, Y 95.3197, Z -5.5000, A 0.000, B 0.000, C 0.000 }
gfCNCPoint4[12074] = {X 121.7854, Y 94.5534, Z -5.5000, A 0.000, B 0.000, C 0.000 }
gfCNCPoint4[12075] = {X 122.4148, Y 93.9095, Z -5.5000, A 0.000, B 0.000, C 0.000 }
gfCNCPoint4[12076] = {X 123.1701, Y 93.4193, Z -5.5000, A 0.000, B 0.000, C 0.000 }
gfCNCPoint4[12077] = {X 124.0145, Y 93.1068, Z -5.5000, A 0.000, B 0.000, C 0.000 }
gfCNCPoint4[12078] = {X 124.9069, Y 92.9870, Z -5.5000, A 0.000, B 0.000, C 0.000 }
gfCNCPoint4[12079] = {X 124.9300, Y 92.9714, Z -5.5000, A 0.000, B 0.000, C 0.000 }
gfCNCPoint4[12080] = {X 124.9630, Y 92.9585, Z -5.5000, A 0.000, B 0.000, C 0.000 }
gfCNCPoint4[12081] = {X 125.4829, Y 92.8814, Z -5.5000, A 0.000, B 0.000, C 0.000 }
